// Core §2.2 lifecycle family, top tier: modes + cascade (§3.4/§3.7), Start/Stop
// mapped onto the §6.1 run command (§6 intro), the step chain (_M_SetStep/_M_Await,
// §6.5/§6.9(b)), the stall walk as a PENDING reason with instant rollup on an
// awaited module's Error (§6.9/§8.2), the §8.11.4 profiler wired in, and
// Starved/Blocked derived from the step's time class (§8.11.4(f)/§8.11.3).
// A Unit type overrides _M_Dispatch (its mode chain) + _M_Supports (+ §3.14 hooks).
FUNCTION_BLOCK ABSTRACT FB_UnitBase EXTENDS FB_CompositeModuleBase IMPLEMENTS I_Unit, I_SequenceHost
VAR_INPUT
    DecisionAnswer : INT;              // §6.11: chosen option index (0 = none yet)
    ReqControlOn   : BOOL;             // §9.8 HMI/data request; edge-consumed and access-gated
    ReqControlOff  : BOOL;
    HmiRequest     : ST_HmiRequest;     // §3.10/§14: arguments first, Sequence last
    {attribute 'OPC.UA.DA' := '0'}
    ControlDomain  : ST_ControlDomainStatus; // §9.8: optional shared cell/cage arrangement
END_VAR
VAR_OUTPUT
    Starved : BOOL;                    // §8.11.3 — derived from CurrentStep.TimeClass
    Blocked : BOOL;
    Domain  : ST_ControlDomainStatus;  // §9.8 read-only publication of the assigned domain
    ControlOnRequest  : BOOL;          // one-scan request to the owning domain coordinator
    ControlOffRequest : BOOL;
END_VAR
VAR_OUTPUT
    Profiler    : FB_CycleProfiler;    // §8.11.4 — HMI chart source
    CurrentStep : ST_StepRecord;       // §6.5 — feeds §6.9 walk AND the profiler
    // §3.13 sequence flow chart. Discovered from _M_SetStep, so a chain author
    // writes nothing; SequenceStepCount is the published length (§8.4 bounded).
    SequenceSteps : ARRAY[1..PL_Fraktal.MAX_SEQUENCE_STEPS] OF ST_SequenceStep;
    // §3.10.2 — the static half of each row: discovered once, never changes, so it
    // stays OFF the cyclic tree and is served through the config manifest under the
    // SAME browse paths as the live half (M_AppendConfig below).
    {attribute 'OPC.UA.DA' := '0'}
    SequenceStepDef : ARRAY[1..PL_Fraktal.MAX_SEQUENCE_STEPS] OF ST_SequenceStepDef;
    // §3.13 — which row each concurrent leg is running. Indexed by branch (0 = the
    // main line), so it is ~10 entries however long the chain is, and cheap enough
    // to stay in the cyclic read: the chart is right the moment its tab opens.
    ActiveSteps : ARRAY[0..PL_Fraktal.MAX_PARALLEL_BRANCHES] OF ST_SequenceCursor;
    // §6.9 — the errors and messages currently attached to rows. Sparse, so a small
    // table instead of 633 bytes reserved on every row for the usually-empty case.
    SequenceAnnotations : ARRAY[1..PL_Fraktal.MAX_SEQUENCE_ANNOTATIONS] OF ST_SequenceAnnotation;
    SequenceAnnotationCount : INT;
    SequenceStepCount : INT;
    CurrentStepElapsed : TIME;         // how long the active step has been running
    CurrentStepTimedOut : BOOL;        // active step outran its guard (§6.9 stall)

    Pending     : ST_Diagnostic;       // live stall reason (Low) — NOT a fault (§6.9)
    Decision    : ST_DecisionRequest;  // §6.11 active request ('' Prompt = none)
    {attribute 'OPC.UA.DA' := '0'}
    StallTime   : TIME := T#30S;       // guard when the step declares no ExpectedTime
    Model       : ST_ModelId;          // §3.1b active model identity (published for HMI/MES/trace)
    // §3.10.2 — static catalogs served via the QUERY_CONFIG manifest, not cyclically
    {attribute 'OPC.UA.DA' := '0'}
    AvailableModelCount : INT;         // §3.8 optional discoverable model/recipe catalog
    {attribute 'OPC.UA.DA' := '0'}
    AvailableModels : ARRAY[1..PL_Fraktal.MAX_RECIPES] OF ST_ModelId;
    Part        : ST_PartContext;      // §3.16.1 live part context (Present=FALSE, Uid='' = none)
    AlarmLog    : FB_AlarmLog;         // §8.3 — active list + closed ring + Blocking
    HostEvents  : FB_HostEventPublisher; // §11.6 fixed, bounded L3/MES projection
    Access      : FB_AccessManager;    // §7.7 — per-root session/policy (default: fully open)
    GoodCount   : UDINT;               // §8.11.2 — cycle verdict counters
    NokCount    : UDINT;
    ReworkCount : UDINT;
    NokReason   : E_Reason;            // §8.11.2 — last NOK's first-out attribution
    MachineState : E_MachineState;     // §8.11.3 — classified every scan (OEE/PackML/host)
    History     : ARRAY[1..PL_Fraktal.MAX_DIAG_RING] OF ST_Diagnostic;  // §6.9(a) ring (newest at HistoryHead)
    HistoryHead : INT;
    {attribute 'OPC.UA.DA' := '0'}
    ModePolicy  : ARRAY[0..PL_Fraktal.MODE_COUNT-1] OF ST_ModePolicy;    // §3.4.1 per-mode switch policy (station cfg; manifest-served)
    RunStyle    : E_RunStyle;          // §3.4.2 active run style (HMI-selectable; CONTINUOUS default)
    Oee         : ST_Oee;              // §8.5.1 accumulators + snapshot (published)
    // §8.5.2 - shifts, when a line is referenced (SetLine). 0 = no shift accounting.
    CurrentShift          : INT;
    ShiftStartedAt        : DT;
    ShiftHistory          : ARRAY[1..PL_Fraktal.MAX_SHIFT_HISTORY] OF ST_ShiftRecord; // newest first
    ShiftHistoryCount     : INT;
    ShiftHistoryTruncated : BOOL;
    OeeTrend    : ARRAY[1..PL_Fraktal.MAX_OEE_SAMPLES] OF ST_OeeSample; // §8.5.1 ring
    OeeTrendHead: INT;                 // newest sample index (0 = none yet)
    HmiResponse : ST_HmiResponse;
    ConfigRev   : UDINT;                // §3.10.2 manifest revision — HMI refetches on change
    // §3.8b — is this station's configuration actually SAFE? Transport
    // acknowledgement and Accepted mean a value is LIVE; this says whether it is
    // DURABLE, whether anything was lost at the last restart, and what the last
    // set operation did. Published cyclically because the answer changes without
    // anybody asking, and because it has to be visible BEFORE the restart that
    // would otherwise reveal it.
    ConfigPersist : ST_ConfigPersistStatus;
    // §3.8b — the store's set listing, refreshed on a LIST_CONFIG_SETS request.
    // Published, and read ON DEMAND: a client target-reads it when a set dialog
    // opens, never in its cyclic snapshot (§1.1 O4). It was marked DA := '0' until
    // 2026-09-27, which made the listing and the export lines unreachable over OPC
    // UA altogether - a client could request them and never read the answer.
    ConfigSets : ARRAY[1..PL_Fraktal.MAX_CONFIG_SETS] OF ST_ConfigSetInfo;
    ConfigSetCount : INT;
    // §3.8b — one line of a set's JSON document, served by EXPORT_CONFIG_SET.
    // Line 0 is the header and 1..RecordCount are the records, so a client pulls
    // a movable document a line at a time without a full buffer in the PLC —
    // the same paging discipline QUERY_CONFIG already uses.
    ConfigSetDocument : STRING(480);
    ConfigSetDocumentLine : INT;
    ConfigSetDocumentLines : INT;
    ModeActivePublished : E_Mode;       // properties are not OPC UA-visible
    RunningPublished : BOOL;
    StopPendingPublished : BOOL;
    SupportedModesPublished : ARRAY[0..PL_Fraktal.MODE_COUNT-1] OF BOOL;
    SupportedRunStylesPublished : ARRAY[0..2] OF BOOL;
    SystemHealth : ST_SystemHealthStatus; // §2.7/§8.12 live, trendable health
    SignalTower  : ST_SignalTowerOut;     // §8.13 single reusable mapping
END_VAR
VAR PERSISTENT
    // §3.8a station-config backing for the manifest-served ModePolicy output.
    // Version 0/unrecognized initializes safe defaults exactly once.
    _modePolicyVersion : UINT;
    _modePolicyStored : ARRAY[0..PL_Fraktal.MODE_COUNT-1] OF ST_ModePolicy;
END_VAR
VAR
    _fTrig    : R_TRIG;
    _mode     : E_Mode;
    _modeReq  : E_Mode;
    _modePend : BOOL;
    _modeExitFirst : BOOL;
    _stopReq  : BOOL;
    {attribute 'OPC.UA.DA' := '0'}
    _awaits   : I_Module;              // module the current step awaits (0 = none)
    _faultEvt : INT;                   // open ERROR event slot in AlarmLog (0 = none)
    _tStall   : TON;
    _seqIndex : INT;                   // row recorded LAST, i.e. the step action running now
    _stepSinceMs : DWORD;              // monotonic start of the main-line step
    // §6.12 — per-row clock and liveness. With a parallel step several rows are
    // active at once, so one cursor is no longer enough to say what is running or
    // for how long. Bounded exactly like the row table itself (§1.1 O10).
    // Per-LEG, not per row: a leg has one active step, so the per-scan sweep is ~10
    // iterations instead of up to MAX_SEQUENCE_STEPS.
    _branchSinceMs : ARRAY[0..PL_Fraktal.MAX_PARALLEL_BRANCHES] OF DWORD;
    _branchTouched : ARRAY[0..PL_Fraktal.MAX_PARALLEL_BRANCHES] OF BOOL;
    _tDecision: TON;                   // §6.11 monotonic active-decision timeout
    _decisionConflictLogged : BOOL;    // one audit record per conflicting request
    _decisionResolutionLogged : BOOL;  // operator/timeout resolution logged once
    _stepReq  : BOOL;                  // §3.4.2 pending single-step request (edge-consumed)
    _holdRun  : BOOL;                  // §3.4.2 HOLD_TO_RUN input held (NON-SAFETY, §9)
    _stepArm  : R_TRIG;
    _errClr   : R_TRIG;                // §6.9 the ERROR state ended
    _oeeLast  : TIME;                  // §8.5.1 last accumulation stamp
    _oeeSampMs: UDINT;                 // ms since last trend sample
    // §8.5.2 shift accounting
    {attribute 'OPC.UA.DA' := '0'}
    _pLine : POINTER TO FB_LineData;
    // §3.8a - model data: the provider and key of this root's own recipe record,
    // and the buffer a model-scoped request loads another model's record into.
    {attribute 'OPC.UA.DA' := '0'}
    _modelProvider : I_RecipeProvider;
    _modelKey : STRING(80);
    _viewModelCode : STRING(64);
    {attribute 'OPC.UA.DA' := '0'}
    _modelBuf : ARRAY[1..PL_Fraktal.MAX_MODEL_DATA_BYTES] OF BYTE;
    _lineHost : BOOL;                  // §3.8e this root ticks the line it references
    _lineRevSeen : UDINT;              // §3.8e line revision last reflected in ConfigRev
    _shiftInit : BOOL;
    _shiftSync : BOOL;
    _shiftManualReset : BOOL;
    _hmiLastSequence : UDINT;
    {attribute 'OPC.UA.DA' := '0'}
    _configPager : FB_ConfigPager;     // §3.10.2 QUERY_CONFIG window writer
    // §3.8b — the parameter-set store. Absent (the shipped default for a Unit
    // nobody wired one into) means save/load/list are simply not offered, which
    // is published as StorePresent = FALSE rather than failing at the first
    // request an operator makes.
    {attribute 'OPC.UA.DA' := '0'}
    _configStore : I_ConfigStore;
    // §3.8b durability. _persistWriter is the shipped LOCAL_RETAIN default and
    // is used unless a deployment injects something else, so a conforming
    // station persists its parametrization with no file system, no network and
    // no configuration — and with no line of project code either (§1.1 O1).
    {attribute 'OPC.UA.DA' := '0'}
    _persistWriter : FB_PersistentDataWriter;
    {attribute 'OPC.UA.DA' := '0'}
    _persistence : I_ConfigPersistence;
    _persistSinceMs : DWORD;           // monotonic ms the current window started at
    _persistEvt : INT;                 // open PersistFailed event slot (0 = none)
    _restoreEvt : INT;                 // open restore-loss event slot (0 = none)
    {attribute 'OPC.UA.DA' := '0'}
    _setJson : FB_ConfigSetJson;       // §3.8b text projection (export/import)
    _importOpen : BOOL;                // an IMPORT_CONFIG_SET save is in progress
    // §3.8b - a set line arriving in pieces (IMPORT_CONFIG_SET, IntValue = 1).
    // A request carries 255 characters and a line may hold 480, so the HMI
    // splits it; the pieces are joined here, and nowhere else.
    {attribute 'OPC.UA.DA' := '0'}
    _importPart : STRING(480);
    // §7.6.1a hold-to-run. The request is LATCHED and re-asserted every scan,
    // because a mailbox delivers one request per sequence and the axis expects
    // to be asked every scan it should keep moving. The latch is what makes
    // that work over a transport; the deadline is what keeps it safe, since a
    // client that stops refreshing - closed, crashed, unplugged - lets the hold
    // expire instead of leaving the machine moving.
    _heldPath  : STRING(255);
    _heldValue : DINT;
    _heldActive : BOOL;
    _heldSinceMs : DWORD;
    // §3.13 - the flow chart changed and the manifest revision owes it a bump.
    // Held until the growth settles, so one burst of row discovery costs one
    // refetch instead of one per row (PL_Fraktal.CHART_REV_SETTLE_MS).
    _chartDirty : BOOL;
    _chartTouchedMs : DWORD;
    {attribute 'OPC.UA.DA' := '0'}
    _carrier  : I_PartCarrier;         // §3.16.2 injected part carrier (0 = traceability off)
    {attribute 'OPC.UA.DA' := '0'}
    _healthPublisher : FB_SystemHealthPublisher;
    {attribute 'OPC.UA.DA' := '0'}
    _healthInput : ST_SystemHealthInput;
    {attribute 'OPC.UA.DA' := '0'}
    _healthParCfg : ST_SystemHealthParCfg;
    _healthConfigured : BOOL;
    {attribute 'OPC.UA.DA' := '0'}
    _towerMapper : FB_SignalTower;
    {attribute 'OPC.UA.DA' := '0'}
    _towerParCfg : ST_SignalTowerParCfg;
    _lampTestRequest : BOOL;
    {attribute 'OPC.UA.DA' := '0'}
    _sequences : ARRAY[1..PL_Fraktal.MAX_SEQUENCES] OF I_Sequence;
    _sequenceCount : INT;
    // §7.5 commissioning/engineering gate register, injected by the composition
    // root. Absent (the shipped default) = a production image: no gate is
    // annunciated and ForceChannel refuses every request (fail closed).
    {attribute 'OPC.UA.DA' := '0'}
    _engineering : REFERENCE TO FB_EngineeringMode;
    // §7.5.2 open standing event per registered gate (0 = none open yet)
    _engineeringEvt : ARRAY[1..PL_Fraktal.MAX_ENGINEERING_GATES] OF INT;
END_VAR
VAR CONSTANT
    // §3.8b — layout version of the retained ModePolicy image. Bump it when a
    // member is added to ST_ModePolicy or the array is resized; the retained
    // image is then rejected and annunciated instead of read by field position.
    MODE_POLICY_SCHEMA : UINT := 1;
    // §3.8b — schema version stamped into every set this root produces, so a set
    // document that outlives the build that wrote it can be recognized rather
    // than guessed at (§13).
    CONFIG_SET_SCHEMA : UINT := 1;
END_VAR

Cyclic();

// Core §7.8 helper — append one non-interlock reason (bounds-checked).
METHOD PROTECTED _M_AddReason
VAR_IN_OUT
    Report : ST_ReleaseReport;
END_VAR
VAR_INPUT
    Text : STRING(255);
    Reason : E_Reason;
    Kind : E_ReleaseKind;
END_VAR
IF Report.Count >= PL_Fraktal.MAX_RELEASE_REASONS THEN
    RETURN;
END_IF
Report.Count := Report.Count + 1;
Report.Reasons[Report.Count].Description := Text;
Report.Reasons[Report.Count].ReasonCode  := Reason;
Report.Reasons[Report.Count].SourcePath  := _name;
Report.Reasons[Report.Count].Kind        := Kind;
Report.Reasons[Report.Count].Bypassable  := FALSE;
END_METHOD

// Core §7.8 — concrete Units override to append the active mode's immediate
// entry/frontier records via PermIntlk.AppendFailed(SourcePath, Report). Future step waits
// stay in CurrentStep/Pending and are not blanket Start conditions. Base: nothing.
METHOD PROTECTED _M_AppendInterlocks
VAR_IN_OUT
    Report : ST_ReleaseReport;
END_VAR
;
END_METHOD

// Core §7.8 — target-aware hook for the MANUAL release rollup: a concrete Unit
// overrides to append the §7.6 Release<Function> conditions of the SPECIFIC target
// module. Base delegates to the Unit-level hook (non-breaking default).
METHOD PROTECTED _M_AppendManualInterlocks
VAR_INPUT
    TargetPath : STRING(255);
    Value : DINT;
END_VAR
VAR_IN_OUT
    Report : ST_ReleaseReport;
END_VAR
_M_AppendInterlocks(Report := Report);
END_METHOD

// §6.11 option-aware release seam. The base validates session, active prompt and
// option identity; a concrete Unit appends the ordinary process conditions that a
// "continue"-style option must satisfy. Safety and child interlocks still remain
// authoritative at their owning modules.
METHOD PROTECTED _M_AppendDecisionInterlocks
VAR_INPUT
    Option : INT;
END_VAR
VAR_IN_OUT
    Report : ST_ReleaseReport;
END_VAR
;
END_METHOD

// §6.11 — publish a typed decision request (single active slot)
METHOD PROTECTED _M_AskDecision
VAR_INPUT
    Req : ST_DecisionRequest;
END_VAR
VAR
    candidate : ST_DecisionRequest;
END_VAR
candidate := Req;
IF candidate.SourcePath = '' THEN
    candidate.SourcePath := _name;
END_IF
// A sequence presents the same request every scan while its step waits. That is
// idempotent. A different producer never overwrites the visible active request.
IF Decision.Prompt <> '' THEN
    IF _M_DecisionMatches(Req := candidate) THEN
        RETURN;
    END_IF
    IF NOT _decisionConflictLogged THEN
        _M_LogDecision(EventKey := 'std.audit.decisionOverlapRejected',
            SourcePath := candidate.SourcePath, Option := 0);
        _decisionConflictLogged := TRUE;
    END_IF
    RETURN;
END_IF
IF NOT _M_ValidateDecision(Req := candidate) THEN
    _M_LogDecision(EventKey := 'std.audit.decisionInvalidRejected',
        SourcePath := candidate.SourcePath, Option := candidate.Default);
    _M_Fault(E_Reason.UNSUPPORTED_COMMAND, 'std.error.invalidDecisionRequest');
    RETURN;
END_IF
Decision := candidate;
DecisionAnswer := 0;
_decisionConflictLogged := FALSE;
_decisionResolutionLogged := FALSE;
_tDecision(IN := FALSE);
_M_LogDecision(EventKey := 'std.audit.decisionRequested',
    SourcePath := Decision.SourcePath, Option := 0);
END_METHOD

// Clear the complete public slot and all private latches atomically.
METHOD PRIVATE _M_ClearDecisionState
VAR
    i : INT;
END_VAR
_tDecision(IN := FALSE);
DecisionAnswer := 0;
Decision.Prompt := '';
Decision.Default := 0;
Decision.Timeout := T#0S;
Decision.SourcePath := '';
FOR i := 1 TO PL_Fraktal.MAX_OPTIONS DO
    Decision.Options[i] := '';
END_FOR
_decisionConflictLogged := FALSE;
_decisionResolutionLogged := FALSE;
END_METHOD

// §6.11 one-slot resolver. Operator input wins if it is accepted in the same scan
// the timeout expires; _M_HandleHmiRequest runs immediately before this method.
METHOD PRIVATE _M_DecisionCyclic
IF _exec <> E_ExecState.BUSY THEN
    IF Decision.Prompt <> '' THEN
        _M_LogDecision(EventKey := 'std.audit.decisionWithdrawn',
            SourcePath := Decision.SourcePath, Option := 0);
        _M_ClearDecisionState();
    ELSE
        _tDecision(IN := FALSE);
    END_IF
    RETURN;
END_IF
IF Decision.Prompt = '' THEN
    _tDecision(IN := FALSE);
    RETURN;
END_IF
IF DecisionAnswer <> 0 THEN
    _tDecision(IN := FALSE);
    IF (DecisionAnswer < 1) OR (DecisionAnswer > PL_Fraktal.MAX_OPTIONS) THEN
        _M_LogDecision(EventKey := 'std.audit.decisionAnswerRejected',
            SourcePath := Decision.SourcePath, Option := DecisionAnswer);
        DecisionAnswer := 0;
        RETURN;
    END_IF
    IF Decision.Options[DecisionAnswer] = '' THEN
        _M_LogDecision(EventKey := 'std.audit.decisionAnswerRejected',
            SourcePath := Decision.SourcePath, Option := DecisionAnswer);
        DecisionAnswer := 0;
        RETURN;
    END_IF
    IF NOT _decisionResolutionLogged THEN
        _M_LogDecision(EventKey := 'std.audit.decisionOperatorResolved',
            SourcePath := Decision.SourcePath, Option := DecisionAnswer);
        _decisionResolutionLogged := TRUE;
    END_IF
    RETURN;
END_IF
IF Decision.Timeout <= T#0S THEN
    _tDecision(IN := FALSE);
    RETURN;
END_IF
_tDecision(IN := TRUE, PT := Decision.Timeout);
IF _tDecision.Q THEN
    DecisionAnswer := Decision.Default;             // validated when accepted
    _tDecision(IN := FALSE);
    _M_LogDecision(EventKey := 'std.audit.decisionTimeoutResolved',
        SourcePath := Decision.SourcePath, Option := DecisionAnswer);
    _decisionResolutionLogged := TRUE;
END_IF
END_METHOD

// Full value comparison makes repeated presentation idempotent while treating a
// changed option/default/timeout as a different request that must not overwrite.
METHOD PRIVATE _M_DecisionMatches : BOOL
VAR_INPUT
    Req : ST_DecisionRequest;
END_VAR
VAR
    i : INT;
END_VAR
_M_DecisionMatches := FALSE;
IF (Decision.Prompt <> Req.Prompt)
OR (Decision.Default <> Req.Default)
OR (Decision.Timeout <> Req.Timeout)
OR (Decision.SourcePath <> Req.SourcePath) THEN
    RETURN;
END_IF
FOR i := 1 TO PL_Fraktal.MAX_OPTIONS DO
    IF Decision.Options[i] <> Req.Options[i] THEN
        RETURN;
    END_IF
END_FOR
_M_DecisionMatches := TRUE;
END_METHOD

// Domain audit: request, rejection and resolution are closed MESSAGE events.
METHOD PRIVATE _M_LogDecision
VAR_INPUT
    EventKey : STRING(160);
    SourcePath : STRING(255);
    Option : INT;
END_VAR
VAR
    slot : INT;
    textValue : STRING(255);
    sourceValue : STRING(255);
END_VAR
textValue := EventKey;
IF Option <> 0 THEN
    textValue := CONCAT(textValue, ' option=');
    textValue := CONCAT(textValue, TO_STRING(Option));
END_IF
sourceValue := SourcePath;
IF sourceValue = '' THEN
    sourceValue := _name;
END_IF
slot := AlarmLog.Raise(Reason := E_Reason.NONE, Text := textValue,
    Source := sourceValue, Severity := E_Severity.LOW,
    Category := E_Category.PROCESS, ResetClass := E_ResetClass.AUTO_RESET);
IF slot > 0 THEN
    AlarmLog.Gone(Slot := slot);
END_IF
END_METHOD

// A finite timeout requires a real safe default. An indefinite request may omit
// Default, but every published request still needs at least one selectable option.
METHOD PRIVATE _M_ValidateDecision : BOOL
VAR_INPUT
    Req : ST_DecisionRequest;
END_VAR
VAR
    i : INT;
    hasOption : BOOL;
END_VAR
_M_ValidateDecision := FALSE;
IF (Req.Prompt = '') OR (Req.Timeout < T#0S) THEN
    RETURN;
END_IF
hasOption := FALSE;
FOR i := 1 TO PL_Fraktal.MAX_OPTIONS DO
    IF Req.Options[i] <> '' THEN
        hasOption := TRUE;
    END_IF
END_FOR
IF NOT hasOption THEN
    RETURN;
END_IF
IF (Req.Timeout > T#0S) OR (Req.Default <> 0) THEN
    IF (Req.Default < 1) OR (Req.Default > PL_Fraktal.MAX_OPTIONS) THEN
        RETURN;
    END_IF
    IF Req.Options[Req.Default] = '' THEN
        RETURN;
    END_IF
END_IF
_M_ValidateDecision := TRUE;
END_METHOD

// §6.9(b) — named plain-condition wait; returns the condition so steps read naturally
METHOD PROTECTED _M_Await : BOOL
VAR_INPUT
    Idx   : INT;
    Label : STRING(120);
    Ok    : BOOL;
END_VAR
IF (Idx >= 1) AND (Idx <= PL_Fraktal.MAX_STEP_CONDS) THEN
    CurrentStep.Conds[Idx].Label := Label;
    CurrentStep.Conds[Idx].Ok    := Ok;
END_IF
_M_Await := Ok;
END_METHOD

// §3.7 — offer the mode to child Units; a child may reject (graceful)
METHOD PROTECTED _M_CascadeMode
VAR_INPUT
    Mode : E_Mode;
END_VAR
VAR
    i  : INT;
    iu : I_Unit;
END_VAR
FOR i := 1 TO _nChild DO
    IF _children[i] <> 0 THEN
        IF __QUERYINTERFACE(_children[i], iu) THEN   // [TC3] capability query — TC3 §3.2
            iu.SetMode(Mode);
        END_IF
    END_IF
END_FOR
END_METHOD

METHOD PROTECTED _M_ClearPending
Pending.ReasonCode  := E_Reason.NONE;
Pending.Description := '';
Pending.TimeSynchronized := FALSE;
END_METHOD

// §14.3 security audit for accepted remote mutations. Operational methods may
// additionally emit their domain event (manual action, OEE reset, shelving); this
// record supplies the remote request kind and authenticated user without secrets.
METHOD PROTECTED _M_AuditHmiAccepted
VAR_INPUT
    Kind : E_HmiRequestKind;
    TargetPath : STRING(255);
    Accepted : BOOL;
END_VAR
VAR
    auditable : BOOL;
    auditSlot : INT;
    textValue : STRING(255);
    sourcePath : STRING(255);
END_VAR
IF NOT Accepted THEN
    RETURN;
END_IF
CASE Kind OF
    E_HmiRequestKind.SET_MODE, E_HmiRequestKind.SET_MODEL,
    E_HmiRequestKind.START, E_HmiRequestKind.STOP,
    E_HmiRequestKind.CONTROL_ON, E_HmiRequestKind.CONTROL_OFF,
    E_HmiRequestKind.OPERATOR_RESET, E_HmiRequestKind.DECISION_ANSWER,
    E_HmiRequestKind.MANUAL_COMMAND, E_HmiRequestKind.SET_RUN_STYLE,
    E_HmiRequestKind.STEP_REQUEST, E_HmiRequestKind.SET_HOLD_RUN,
    E_HmiRequestKind.RESET_OEE, E_HmiRequestKind.WRITE_CONFIG,
    E_HmiRequestKind.SHELVE_ALARM, E_HmiRequestKind.UNSHELVE_ALARM,
    E_HmiRequestKind.FORCE_CHANNEL, E_HmiRequestKind.SET_ACCESS_LEVEL,
    E_HmiRequestKind.SET_SESSION_TIMEOUT, E_HmiRequestKind.LAMP_TEST,
    E_HmiRequestKind.CAPTURE_CONFIG, E_HmiRequestKind.SAVE_CONFIG_SET,
    E_HmiRequestKind.LOAD_CONFIG_SET, E_HmiRequestKind.ACK_CONFIG_RESTORE,
    E_HmiRequestKind.IMPORT_CONFIG_SET, E_HmiRequestKind.DELETE_CONFIG_SET,
    E_HmiRequestKind.SET_CLASS_LEVEL:
        auditable := TRUE;
ELSE
    auditable := FALSE;
END_CASE
IF NOT auditable THEN
    RETURN;
END_IF
Access.RecordActivity();
textValue := CONCAT('std.audit.hmiAccepted kind=', TO_STRING(TO_DINT(Kind)));
textValue := CONCAT(textValue, ' user=');
textValue := CONCAT(textValue, Access.CurrentUser);
// §3.8b — a set operation is audited WITH the set name and record count: "the
// operator loaded a set" is not an audit record anyone can act on later.
IF (Kind = E_HmiRequestKind.SAVE_CONFIG_SET)
OR (Kind = E_HmiRequestKind.LOAD_CONFIG_SET)
OR (Kind = E_HmiRequestKind.DELETE_CONFIG_SET) THEN
    textValue := CONCAT(textValue, ' set=');
    textValue := CONCAT(textValue, ConfigPersist.LastSetName);
    textValue := CONCAT(textValue, ' records=');
    textValue := CONCAT(textValue, INT_TO_STRING(ConfigPersist.LastSetRecords));
END_IF
sourcePath := TargetPath;
IF sourcePath = '' THEN
    sourcePath := _name;
END_IF
auditSlot := AlarmLog.Raise(Reason := E_Reason.NONE, Text := textValue,
    Source := sourcePath, Severity := E_Severity.LOW, Category := E_Category.SYSTEM,
    ResetClass := E_ResetClass.AUTO_RESET);
IF auditSlot > 0 THEN AlarmLog.Gone(Slot := auditSlot); END_IF
END_METHOD

// Module paths are qualified dotted Fraktal identities (§4.8). A request routed
// through this root may target the root itself or one descendant, never a peer.
METHOD PRIVATE _M_OwnsModulePath : BOOL
VAR_INPUT
    Path : STRING(255);
END_VAR
VAR
    prefix : STRING(255);
END_VAR
prefix := CONCAT(_name, '.');
_M_OwnsModulePath := (Path = _name) OR (FIND(Path, prefix) = 1);
END_METHOD

// call at the finish step (§8.11.1): publishes the profile; FALSE = stop granted
METHOD PROTECTED _M_EndOfCycle : BOOL
Profiler.CycleComplete();
IF _stopReq THEN
    _stopReq := FALSE;
    Execute := FALSE;
    _M_Complete();
    _M_EndOfCycle := FALSE;
ELSE
    _M_EndOfCycle := TRUE;
END_IF
END_METHOD

// §3.10/§14 — consume one committed OPC UA request exactly once.
METHOD PROTECTED _M_HandleHmiRequest
VAR
    modelId  : ST_ModelId;
    modeReq  : E_Mode;
    styleReq : E_RunStyle;
    gateReq  : E_GatedAction;
    levelReq : E_AccessLevel;
    alarmSlot : INT;
    policyValueValid : BOOL;
    configKindReq : E_ConfigKind;
END_VAR
IF HmiRequest.Sequence = _hmiLastSequence THEN
    RETURN;
ELSE
    _hmiLastSequence := HmiRequest.Sequence;
END_IF

HmiResponse.Accepted := FALSE;
HmiResponse.Diagnostic := '';
HmiResponse.Report.Count := 0;
HmiResponse.Report.Released := FALSE;
// A held line piece belongs to the very next import request. Anything else in
// between means the line was abandoned, so it is dropped rather than glued to
// whatever arrives later.
IF HmiRequest.Kind <> E_HmiRequestKind.IMPORT_CONFIG_SET THEN
    _importPart := '';
END_IF

CASE HmiRequest.Kind OF
    E_HmiRequestKind.LOGIN:
        HmiResponse.Accepted := Access.RequestLogin(User := HmiRequest.User, Secret := HmiRequest.Secret);
    E_HmiRequestKind.LOGOUT:
        HmiResponse.Accepted := Access.RequestLogout();
    E_HmiRequestKind.SET_MODE:
        IF (HmiRequest.IntValue >= 0) AND (HmiRequest.IntValue < PL_Fraktal.MODE_COUNT) THEN
            modeReq := HmiRequest.IntValue;
            HmiResponse.Accepted := SetMode(Mode := modeReq);
        ELSE
            HmiResponse.Diagnostic := 'std.error.unsupportedModeRequest';
        END_IF
    E_HmiRequestKind.SET_MODEL:
        modelId.ModelCode := HmiRequest.TextValue;
        HmiResponse.Accepted := SetModel(Id := modelId);
    E_HmiRequestKind.START:
        HmiResponse.Accepted := Start();
    E_HmiRequestKind.STOP:
        HmiResponse.Accepted := Stop();
    E_HmiRequestKind.CONTROL_ON:
        HmiResponse.Accepted := RequestControlPower(ControlOn := TRUE);
    E_HmiRequestKind.CONTROL_OFF:
        HmiResponse.Accepted := RequestControlPower(ControlOn := FALSE);
    E_HmiRequestKind.OPERATOR_RESET:
        HmiResponse.Accepted := OperatorReset();
    E_HmiRequestKind.DECISION_ANSWER:
        HmiResponse.Accepted := SubmitDecision(Option := TO_INT(HmiRequest.IntValue),
            Report := HmiResponse.Report);
    E_HmiRequestKind.MANUAL_COMMAND:
        HmiResponse.Accepted := ManualCommandTo(TargetPath := HmiRequest.TargetPath, Value := HmiRequest.IntValue);
    E_HmiRequestKind.MANUAL_HELD:
        HmiResponse.Accepted := ManualHeldTo(TargetPath := HmiRequest.TargetPath,
            Value := HmiRequest.IntValue, Held := HmiRequest.BoolValue);
    E_HmiRequestKind.SET_RUN_STYLE:
        IF (HmiRequest.IntValue >= 0) AND (HmiRequest.IntValue <= 2) THEN
            styleReq := HmiRequest.IntValue;
            HmiResponse.Accepted := SetRunStyle(Style := styleReq);
        ELSE
            HmiResponse.Diagnostic := 'std.error.unsupportedRunStyleRequest';
        END_IF
    E_HmiRequestKind.STEP_REQUEST:
        HmiResponse.Accepted := StepRequest();
    E_HmiRequestKind.SET_HOLD_RUN:
        HmiResponse.Accepted := SetHoldRun(Held := HmiRequest.BoolValue);
    E_HmiRequestKind.RELEASE_START:
        ReleaseReportStart(Report := HmiResponse.Report);
        HmiResponse.Accepted := TRUE;
    E_HmiRequestKind.RELEASE_MANUAL:
        ReleaseReportManual(TargetPath := HmiRequest.TargetPath, Value := HmiRequest.IntValue,
            Report := HmiResponse.Report);
        HmiResponse.Accepted := TRUE;
    E_HmiRequestKind.RELEASE_ACTION:
        IF (HmiRequest.IntValue >= 0)
        AND (HmiRequest.IntValue <= TO_DINT(E_GatedAction.CONFIG_SET)) THEN
            gateReq := HmiRequest.IntValue;
            ReleaseReportAction(Gate := gateReq, Report := HmiResponse.Report);
            HmiResponse.Accepted := TRUE;
        ELSE
            HmiResponse.Diagnostic := 'std.error.unsupportedGatedActionRequest';
        END_IF
    E_HmiRequestKind.RESET_OEE:
        HmiResponse.Accepted := ResetOee();
    E_HmiRequestKind.WRITE_CONFIG:
        // §3.8a - DurationMs names the model a model-data write is for
        // (0 = the active model, n = AvailableModels[n]); other values ignore it.
        HmiResponse.Accepted := WriteModelConfig(ModelIndex := HmiRequest.DurationMs,
            TargetPath := HmiRequest.TargetPath, WriteKey := HmiRequest.NameValue,
            Revision := HmiRequest.IntValue, TextValue := HmiRequest.TextValue);
    E_HmiRequestKind.SHELVE_ALARM:
        alarmSlot := AlarmLog.FindActiveSlot(SourcePath := HmiRequest.TargetPath,
            Description := HmiRequest.TextValue);
        IF alarmSlot > 0 THEN
            HmiResponse.Accepted := ShelveAlarm(Slot := alarmSlot,
                DurationS := HmiRequest.DurationMs / 1000);
        ELSE
            HmiResponse.Diagnostic := 'std.error.alarmIdentityNotUnique';
        END_IF
    E_HmiRequestKind.UNSHELVE_ALARM:
        alarmSlot := AlarmLog.FindActiveSlot(SourcePath := HmiRequest.TargetPath,
            Description := HmiRequest.TextValue);
        IF alarmSlot > 0 THEN
            HmiResponse.Accepted := UnshelveAlarm(Slot := alarmSlot);
        ELSE
            HmiResponse.Diagnostic := 'std.error.alarmIdentityNotUnique';
        END_IF
    E_HmiRequestKind.FORCE_CHANNEL:
        HmiResponse.Accepted := ForceChannel(ChannelPath := HmiRequest.TargetPath,
            Force := HmiRequest.BoolValue, BoolText := HmiRequest.TextValue,
            AnalogText := HmiRequest.NameValue);
    E_HmiRequestKind.QUERY_CONFIG:
        // §3.10.2 — serve one manifest page: re-walk the deterministic export
        // enumeration, storing only the requested window (no full buffer).
        // §3.8d: no blanket DATA_READ refusal any more - a class may be readable
        // below it. Each entry is served with or without its value by its level.
        _configPager.M_SetAccess(pAccess := ADR(Access));
        // §3.8a - DurationMs names the model whose model-data values to serve.
        IF NOT _configPager.M_Setup(Target := ADR(HmiResponse.ConfigPage),
            PageIndex := TO_INT(HmiRequest.IntValue), Revision := ConfigRev) THEN
            HmiResponse.Diagnostic := 'std.error.hmiRequestRejected';
        ELSIF M_AppendModelConfig(Pager := _configPager,
                ModelIndex := HmiRequest.DurationMs) THEN
            _configPager.M_Finish();
            HmiResponse.Accepted := TRUE;
        ELSE
            HmiResponse.Diagnostic := 'std.error.modelNotAvailable';
        END_IF
    E_HmiRequestKind.SET_ACCESS_LEVEL:
        policyValueValid := TRUE;
        IF HmiRequest.TextValue = '0' THEN
            levelReq := E_AccessLevel.NONE;
        ELSIF HmiRequest.TextValue = '1' THEN
            levelReq := E_AccessLevel.OPERATOR;
        ELSIF HmiRequest.TextValue = '2' THEN
            levelReq := E_AccessLevel.TECHNICIAN;
        ELSIF HmiRequest.TextValue = '3' THEN
            levelReq := E_AccessLevel.ENGINEER;
        ELSIF HmiRequest.TextValue = '4' THEN
            levelReq := E_AccessLevel.ADMIN;
        ELSE
            policyValueValid := FALSE;
        END_IF
        IF policyValueValid
        AND (HmiRequest.IntValue >= 0)
        AND (HmiRequest.IntValue <= TO_DINT(E_GatedAction.CONFIG_SET)) THEN
            gateReq := HmiRequest.IntValue;
            HmiResponse.Accepted := SetAccessLevel(Gate := gateReq, Level := levelReq);
        ELSE
            HmiResponse.Diagnostic := 'std.error.accessPolicyValueInvalid';
        END_IF
    E_HmiRequestKind.SET_SESSION_TIMEOUT:
        HmiResponse.Accepted := SetSessionTimeout(TimeoutMs := HmiRequest.DurationMs);
    E_HmiRequestKind.LAMP_TEST:
        HmiResponse.Accepted := RequestLampTest();
    E_HmiRequestKind.CAPTURE_CONFIG:
        // §3.8c(a) — a capture is routed through the SAME acknowledged mailbox as
        // the typed write it replaces, with the same arguments minus the value:
        // the number comes from the machine, not from the client.
        HmiResponse.Accepted := CaptureConfig(TargetPath := HmiRequest.TargetPath,
            WriteKey := HmiRequest.NameValue, Revision := HmiRequest.IntValue);
    E_HmiRequestKind.SAVE_CONFIG_SET:
        IF (HmiRequest.IntValue >= 0)
        AND (HmiRequest.IntValue <= TO_DINT(E_ConfigKind.LINE_CFG)) THEN
            configKindReq := HmiRequest.IntValue;
            HmiResponse.Accepted := SaveConfigSet(SetName := HmiRequest.TextValue,
                Kind := configKindReq);
        ELSE
            HmiResponse.Diagnostic := 'std.error.configSetKindInvalid';
        END_IF
    E_HmiRequestKind.LOAD_CONFIG_SET:
        HmiResponse.Accepted := LoadConfigSet(SetName := HmiRequest.TextValue);
        IF NOT HmiResponse.Accepted THEN
            HmiResponse.Diagnostic := 'std.error.configSetRejected';
        END_IF
    E_HmiRequestKind.LIST_CONFIG_SETS:
        HmiResponse.Accepted := ListConfigSets();
    E_HmiRequestKind.ACK_CONFIG_RESTORE:
        HmiResponse.Accepted := AcknowledgeConfigRestore();
        IF NOT HmiResponse.Accepted THEN
            HmiResponse.Diagnostic := 'std.error.configRestoreAckRefused';
        END_IF
    E_HmiRequestKind.EXPORT_CONFIG_SET:
        HmiResponse.Accepted := ExportConfigSetLine(SetName := HmiRequest.TextValue,
            Line := TO_INT(HmiRequest.IntValue));
    E_HmiRequestKind.IMPORT_CONFIG_SET:
        HmiResponse.Accepted := ImportConfigSetPiece(Piece := HmiRequest.TextValue,
            More := HmiRequest.IntValue = 1, Commit := HmiRequest.BoolValue);
        IF NOT HmiResponse.Accepted THEN
            HmiResponse.Diagnostic := 'std.error.configSetLineRejected';
        END_IF
    E_HmiRequestKind.SET_CLASS_LEVEL:
        HmiResponse.Accepted := SetDataClassLevel(ClassId := HmiRequest.NameValue,
            Level := HmiRequest.IntValue, ForWrite := HmiRequest.BoolValue);
        IF NOT HmiResponse.Accepted THEN
            HmiResponse.Diagnostic := 'std.error.accessPolicyValueInvalid';
        END_IF
    E_HmiRequestKind.DELETE_CONFIG_SET:
        HmiResponse.Accepted := DeleteConfigSet(SetName := HmiRequest.TextValue);
        IF NOT HmiResponse.Accepted THEN
            HmiResponse.Diagnostic := 'std.error.configSetDeleteRefused';
        END_IF
    E_HmiRequestKind.NONE:
        HmiResponse.Diagnostic := 'std.error.emptyHmiRequest';
ELSE
    HmiResponse.Diagnostic := 'std.error.unsupportedHmiRequest';
END_CASE

IF NOT HmiResponse.Accepted AND (HmiResponse.Diagnostic = '') THEN
    HmiResponse.Diagnostic := 'std.error.hmiRequestRejected';
ELSE
    HmiResponse.Diagnostic := HmiResponse.Diagnostic;
END_IF
_M_AuditHmiAccepted(Kind := HmiRequest.Kind, TargetPath := HmiRequest.TargetPath,
    Accepted := HmiResponse.Accepted);
HmiRequest.Secret := '';
HmiResponse.AckSequence := _hmiLastSequence;
END_METHOD

// §11.6 one owning projection helper; callers supply only event-specific fields.
METHOD PRIVATE _M_HostEvent : BOOL
VAR_INPUT
    Kind          : E_HostEventKind;
    PartUid       : STRING(64);
    Subject       : STRING(80);
    Value         : STRING(80);
    Verdict       : E_Verdict;
    ReasonCode    : E_Reason;
END_VAR
_M_HostEvent := HostEvents.Emit(Kind := Kind,
    StationPath := _name, PartUid := PartUid, Subject := Subject,
    Value := Value, Verdict := Verdict, ReasonCode := ReasonCode);
END_METHOD

// §3.4.1/§3.14.4 — default per-mode switch policy. Station config (§3.8a) may
// overwrite ModePolicy[] after this. By FRAMEWORK DEFAULT a mode change while a
// sequence runs performs an IMMEDIATE software abort (E-stop-like, not a safety
// function, §3.14.4) — so Style defaults to IMMEDIATE. GRACEFUL completion is an
// opt-in: a Unit overrides OnModeExit to stop-after-cycle, or station config sets
// Style := GRACEFUL for a mode. Shield only governs acceptance while running.
METHOD PROTECTED _M_InitModePolicy
VAR
    i : INT;
END_VAR
FOR i := 0 TO PL_Fraktal.MODE_COUNT-1 DO
    ModePolicy[i].Shield := E_ModeSwitchShield.CONFIRM;
    ModePolicy[i].Style  := E_ModeSwitchStyle.IMMEDIATE;
END_FOR
// Setup modes a running machine may not leave without an explicit Stop first.
ModePolicy[TO_INT(E_Mode.CHANGEOVER)].Shield := E_ModeSwitchShield.BLOCKED_WHILE_RUNNING;
ModePolicy[TO_INT(E_Mode.CALIBRATION)].Shield:= E_ModeSwitchShield.BLOCKED_WHILE_RUNNING;
// HOME and MANUAL are freely interruptible; both inherit the IMMEDIATE default.
ModePolicy[TO_INT(E_Mode.HOME)].Shield       := E_ModeSwitchShield.INTERRUPTIBLE;
ModePolicy[TO_INT(E_Mode.MANUAL)].Shield     := E_ModeSwitchShield.INTERRUPTIBLE;
END_METHOD

// §8.5.1 — pure recompute of A/P/Q/OEE from the accumulators (testable in isolation).
// Invalid factors are OMITTED from the product, never assumed 100% (O7).
METHOD PROTECTED _M_OeeCompute
VAR
    total : UDINT;
    denomA: UDINT;
END_VAR
denomA := Oee.RunMs + Oee.DownMs;
Oee.AvailValid := denomA > 0;
IF Oee.AvailValid THEN
    Oee.Availability := UDINT_TO_REAL(Oee.RunMs) / UDINT_TO_REAL(denomA);
ELSE
    Oee.Availability := 0.0;
END_IF
Oee.PerfValid := (Oee.IdealCycleMs > 0) AND (Oee.RunMs > 0);
IF Oee.PerfValid THEN
    Oee.Performance := UDINT_TO_REAL(Oee.IdealCycleMs) * UDINT_TO_REAL(GoodCount + NokCount)
                       / UDINT_TO_REAL(Oee.RunMs);
    IF Oee.Performance > 1.0 THEN
        Oee.Performance := 1.0;          // faster than ideal caps at 100% (standard practice)
    END_IF
ELSE
    Oee.Performance := 0.0;
END_IF
total := GoodCount + NokCount;
Oee.QualValid := total > 0;
IF Oee.QualValid THEN
    Oee.Quality := UDINT_TO_REAL(GoodCount) / UDINT_TO_REAL(total);
ELSE
    Oee.Quality := 0.0;
END_IF
// product of VALID factors only; OEE valid iff at least one factor is valid
Oee.Oee := 1.0;
Oee.OeeValid := FALSE;
IF Oee.AvailValid THEN Oee.Oee := Oee.Oee * Oee.Availability; Oee.OeeValid := TRUE; END_IF
IF Oee.PerfValid  THEN Oee.Oee := Oee.Oee * Oee.Performance;  Oee.OeeValid := TRUE; END_IF
IF Oee.QualValid  THEN Oee.Oee := Oee.Oee * Oee.Quality;      Oee.OeeValid := TRUE; END_IF
IF NOT Oee.OeeValid THEN
    Oee.Oee := 0.0;
END_IF
END_METHOD

// §8.5.1 — attribute elapsed time to run/down/idle, recompute factors, sample ring.
METHOD PROTECTED _M_OeeUpdate
VAR
    currentTime : TIME;
    deltaMs     : UDINT;
END_VAR
currentTime := TIME();                 // monotonic duration clock
IF _oeeLast = T#0S THEN
    _oeeLast := currentTime;
    RETURN;
END_IF
deltaMs := TIME_TO_UDINT(currentTime) - TIME_TO_UDINT(_oeeLast); // wrap-safe on UDINT subtraction
_oeeLast := currentTime;
IF _exec = E_ExecState.BUSY THEN
    Oee.RunMs := Oee.RunMs + deltaMs;
ELSIF (_exec = E_ExecState.ERROR) OR AlarmLog.Blocking THEN
    Oee.DownMs := Oee.DownMs + deltaMs;
ELSE
    Oee.IdleMs := Oee.IdleMs + deltaMs;
END_IF
_M_OeeCompute();
_oeeSampMs := _oeeSampMs + deltaMs;
IF _oeeSampMs >= PL_Fraktal.OEE_SAMPLE_MS THEN
    _oeeSampMs := 0;
    OeeTrendHead := (OeeTrendHead MOD PL_Fraktal.MAX_OEE_SAMPLES) + 1;
    OeeTrend[OeeTrendHead].Availability := Oee.Availability;
    OeeTrend[OeeTrendHead].Performance  := Oee.Performance;
    OeeTrend[OeeTrendHead].Quality      := Oee.Quality;
    OeeTrend[OeeTrendHead].Oee          := Oee.Oee;
    OeeTrend[OeeTrendHead].OeeValid     := Oee.OeeValid;
END_IF
END_METHOD

// §3.16.3 EVENT_PART_PROCESSING_ABORTED — the part leaves without a valid result
// (fault, abort, manual removal). Called automatically on Unit ERROR entry.
METHOD PROTECTED _M_PartAborted
IF (_carrier = 0) OR NOT Part.Present THEN
    RETURN;
END_IF
Part.Result.Verdict := E_Verdict.NONE;
IF (_exec = E_ExecState.ERROR) AND (Part.Result.ReasonCode = E_Reason.NONE) THEN
    Part.Result.ReasonCode := _diag.ReasonCode;
END_IF
_M_PartEvent(Reason := E_Reason.EVENT_PART_PROCESSING_ABORTED,
    Text := 'std.event.partAborted: ');
_M_HostEvent(Kind := E_HostEventKind.PROCESSING_ABORTED, PartUid := Part.Uid,
    Subject := '', Value := '',
    Verdict := E_Verdict.NONE, ReasonCode := Part.Result.ReasonCode);
Part.Present := FALSE;
END_METHOD

// §3.16.3 — one canonical part-lifecycle event: instant come+gone MESSAGE ring entry.
METHOD PRIVATE _M_PartEvent
VAR_INPUT
    Reason : E_Reason;
    Text : STRING(255);
END_VAR
VAR
    slot : INT;
    txt : STRING(255);
END_VAR
txt := CONCAT(Text, Part.Uid);
slot := AlarmLog.Raise(Reason := Reason, Text := txt, Source := _name,
    Severity := E_Severity.LOW, Category := E_Category.PROCESS,
    ResetClass := E_ResetClass.AUTO_RESET);
IF slot > 0 THEN
    AlarmLog.Gone(Slot := slot);
END_IF
END_METHOD

// §3.16.3 EVENT_PART_PROCESSED — stamp the verdict, write the carrier FIRST
// (result-before-event contract), then raise the event. The Uid and result stay
// published until the next part so the HMI shows the last outcome.
METHOD PROTECTED _M_PartProcessed : BOOL
VAR_INPUT
    Verdict : E_Verdict;
    Reason : E_Reason;
END_VAR
_M_PartProcessed := FALSE;
IF (_carrier = 0) OR NOT Part.Present THEN
    RETURN;
END_IF
// A reject without a first-out reason cannot satisfy the KPI or host contract.
// Reject it before writing the carrier so result-before-event remains atomic.
IF (Verdict = E_Verdict.NOK) AND (Reason = E_Reason.NONE) THEN
    _M_Fault(E_Reason.RESULT_RECORD_REJECTED, 'std.error.nokReasonRequired');
    RETURN;
END_IF
Part.Result.Verdict := Verdict;
Part.Result.ReasonCode := Reason;
Part.Result.StationPath := _name;
Part.Result.Stamp := F_Now();
Part.Result.TimeSynchronized := F_TimeSynchronized();
IF NOT _carrier.WriteResult(Ctx := Part) THEN
    _M_Fault(E_Reason.CARRIER_WRITE_FAILED, 'std.error.partCarrierWriteFailed');
    RETURN;
END_IF
// §8.11.2 — counters increment HERE, from the verdict; an NOK carries its
// first-out ReasonCode so scrap is analysable by cause (§8.8 vocabulary).
CASE Verdict OF
    E_Verdict.OK:     CountGood();
    E_Verdict.NOK:
        IF NOT CountNok(Reason := Reason) THEN
            RETURN;
        END_IF
    E_Verdict.REWORK: CountRework();
ELSE
    ;                                // NONE: no count — the part left unjudged
END_CASE
_M_PartEvent(Reason := E_Reason.EVENT_PART_PROCESSED, Text := 'std.event.partProcessed: ');
_M_HostEvent(Kind := E_HostEventKind.PROCESSED, PartUid := Part.Uid,
    Subject := '', Value := '',
    Verdict := Verdict, ReasonCode := Reason);
Part.Present := FALSE;
_M_PartProcessed := TRUE;
END_METHOD

// §3.16.3 EVENT_PART_RECEIVED — confirm identity at station entry via the carrier.
// FALSE with a CARRIER_READ_FAILED fault on a failed read (never silent), FALSE
// silently when no carrier is configured (§3.9 feature selectability).
METHOD PROTECTED _M_PartReceived : BOOL
VAR
    i : INT;
END_VAR
_M_PartReceived := FALSE;
IF _carrier = 0 THEN
    RETURN;
END_IF
Part.Uid := '';                              // station entry = fresh identity read
IF NOT _carrier.ReadContext(Ctx := Part) THEN
    _M_Fault(E_Reason.CARRIER_READ_FAILED, 'std.error.partCarrierReadFailed');
    RETURN;
END_IF
Part.Result.Verdict := E_Verdict.NONE;       // this station's outcome starts empty
Part.Result.ReasonCode := E_Reason.NONE;
Part.Result.StationPath := _name;
FOR i := 1 TO PL_Fraktal.MAX_RESULTS DO
    Part.Result.Records[i].Name := '';
END_FOR
_M_PartEvent(Reason := E_Reason.EVENT_PART_RECEIVED, Text := 'std.event.partReceived: ');
_M_HostEvent(Kind := E_HostEventKind.PART_RECEIVED, PartUid := Part.Uid,
    Subject := '', Value := '',
    Verdict := E_Verdict.NONE, ReasonCode := E_Reason.NONE);
_M_PartReceived := TRUE;
END_METHOD

// §3.16.1 — append one measured value to this part's result (test cells).
// FALSE when the bounded record table is full (RESULT_RECORD_REJECTED semantics).
METHOD PROTECTED _M_PartRecord : BOOL
VAR_INPUT
    RecordName : STRING(64);
    Value : LREAL;
    Minimum : LREAL;
    Maximum : LREAL;
    Target : LREAL;
    EngUnit : STRING(16);
END_VAR
VAR
    i : INT;
END_VAR
_M_PartRecord := FALSE;
IF NOT Part.Present THEN
    RETURN;
END_IF
FOR i := 1 TO PL_Fraktal.MAX_RESULTS DO
    IF Part.Result.Records[i].Name = '' THEN
        Part.Result.Records[i].Name := RecordName;
        Part.Result.Records[i].Value := Value;
        Part.Result.Records[i].Minimum := Minimum;
        Part.Result.Records[i].Maximum := Maximum;
        Part.Result.Records[i].Target := Target;
        Part.Result.Records[i].Unit := EngUnit;
        Part.Result.Records[i].InTol := (Maximum <= Minimum)
            OR ((Value >= Minimum) AND (Value <= Maximum));
        _M_PartRecord := TRUE;
        RETURN;
    END_IF
END_FOR
END_METHOD

// §3.16.3 EVENT_PART_PROCESSING_STARTED — the value-adding sequence begins.
METHOD PROTECTED _M_PartStarted
IF (_carrier = 0) OR NOT Part.Present THEN
    RETURN;
END_IF
_M_PartEvent(Reason := E_Reason.EVENT_PART_PROCESSING_STARTED,
    Text := 'std.event.partProcessingStarted: ');
_M_HostEvent(Kind := E_HostEventKind.PROCESSING_STARTED, PartUid := Part.Uid,
    Subject := '', Value := '',
    Verdict := E_Verdict.NONE, ReasonCode := E_Reason.NONE);
END_METHOD

// §6.9/§3.10(a') — overlay the pending stall after the common mirror refresh.
METHOD PROTECTED _M_PublishStatus
SUPER^._M_PublishStatus();
// §8.11.4(f)/§8.11.3 — one declaration, two views. Derived AFTER dispatch so the
// wait class reflects the step record this scan just set, not the previous one.
// §3.13 — live row state for the flow chart: how long the active step has run,
// and whether it outran its declared guard (the same watchdog §6.9 stalls on).
IF _exec = E_ExecState.BUSY THEN
    CurrentStepElapsed := DWORD_TO_TIME(TIME_TO_DWORD(TIME()) - _stepSinceMs);
ELSE
    CurrentStepElapsed := T#0S;
END_IF
CurrentStepTimedOut := _tStall.Q;
Starved := (_exec = E_ExecState.BUSY) AND (CurrentStep.TimeClass = E_TimeClass.WAIT_UPSTREAM);
Blocked := (_exec = E_ExecState.BUSY) AND (CurrentStep.TimeClass = E_TimeClass.WAIT_DOWNSTREAM);
// §8.11.3 — classify into the fixed machine-state set (priority: fault first,
// then planned states, then line attribution, then producing/idle).
IF (_exec = E_ExecState.ERROR) OR AlarmLog.Blocking THEN
    MachineState := E_MachineState.DOWN;
ELSIF _mode = E_Mode.CHANGEOVER THEN
    MachineState := E_MachineState.CHANGEOVER;
ELSIF Blocked THEN
    MachineState := E_MachineState.BLOCKED;
ELSIF Starved THEN
    MachineState := E_MachineState.STARVED;
ELSIF _exec = E_ExecState.BUSY THEN
    MachineState := E_MachineState.PRODUCING;
ELSIF _stopReq OR (_exec = E_ExecState.ABORTED) THEN
    MachineState := E_MachineState.STOPPED;
ELSE
    MachineState := E_MachineState.IDLE;
END_IF
Status.ControlDomainId := ControlDomain.Id;
Domain := ControlDomain;
Safety := ControlDomain.Safety;             // read-only HMI mirror; ownership stays in domain
ControlPower := ControlDomain.ControlPower;
IF (_exec <> E_ExecState.ERROR) AND (Pending.ReasonCode <> E_Reason.NONE) THEN
    Status.Diagnostic := Pending;
END_IF
END_METHOD

// §6.9(a) — fixed ring, newest at HistoryHead; never allocates
METHOD PROTECTED _M_PushHistory
VAR_INPUT
    D : ST_Diagnostic;
END_VAR
HistoryHead := (HistoryHead MOD PL_Fraktal.MAX_DIAG_RING) + 1;
History[HistoryHead] := D;
END_METHOD

// §8.11.4(d)/§8.12 — a Low-severity maintenance event: informs planning, does not
// stop the cycle. Instant come+gone ring entry (the trend data lives in Profiler).
METHOD PROTECTED _M_RaiseMaintenance
VAR_INPUT
    Reason : E_Reason;
    Text : STRING(255);
END_VAR
VAR
    slot : INT;
END_VAR
slot := AlarmLog.Raise(Reason := Reason, Text := Text, Source := _name,
    Severity := E_Severity.LOW, Category := E_Category.SYSTEM,
    ResetClass := E_ResetClass.AUTO_RESET);
IF slot > 0 THEN
    AlarmLog.Gone(Slot := slot);
END_IF
END_METHOD

// §3.8b — route a published editable field to the module that registered it.
// WriteConfig already owns access and root-path checks; the recursive walk finds
// the owner by Scope, and that module rechecks revision, type, range, domain and
// its own invariants before storing. A type whose values are declared through
// M_RegisterConfig* therefore needs no override at all, which is the point: a new
// module type costs no routing code (§1.1 O1). Framework-owned keys never reach
// here — _M_WriteBaseConfig answers those first. An override that adds
// hand-written routing shall call SUPER^ first and keep its own answer only when
// the base declines.
METHOD PROTECTED _M_RouteConfigWrite : BOOL
VAR_INPUT
    TargetPath : STRING(255);
    WriteKey   : STRING(160);
    Revision   : UDINT;
    TextValue  : STRING(255);
END_VAR
// RequiresReady is a question about THIS root's state, which the owning child
// cannot see from where it sits, so the root answers it on the way down.
_M_RouteConfigWrite := M_ApplyConfigWrite(Scope := TargetPath,
    WriteKey := WriteKey, Revision := Revision, TextValue := TextValue,
    // Another model's record is not what the machine is running on.
    RootReady := (_exec = E_ExecState.READY) OR (_pModelView <> 0));
END_METHOD

// Framework-owned typed handlers. Stable keys are independent of browse paths;
// capability revision 1 accepts exact enum ordinals and only while READY.
//
// Commit := FALSE validates and stores nothing — the staging pass of a §3.8b set
// load. The root's own ModePolicy keys are published as STATION_CFG
// capabilities, so they are in every station set and have to stage through the
// same validator that writes them, for the same reason every module's do.
METHOD PRIVATE _M_WriteBaseConfig : BOOL
VAR_INPUT
    TargetPath : STRING(255);
    WriteKey   : STRING(160);
    Revision   : UDINT;
    TextValue  : STRING(255);
    Commit     : BOOL;
END_VAR
VAR
    i      : INT;
    key    : STRING(160);
    shield : E_ModeSwitchShield;
    style  : E_ModeSwitchStyle;
END_VAR
_M_WriteBaseConfig := FALSE;
IF (TargetPath <> Status.Name) OR (Revision <> 1) OR (_exec <> E_ExecState.READY) THEN
    RETURN;
END_IF
FOR i := 0 TO PL_Fraktal.MODE_COUNT - 1 DO
    key := CONCAT('unit.modePolicy.', CONCAT(TO_STRING(i), '.shield'));
    IF WriteKey = key THEN
        IF TextValue = '0' THEN
            shield := E_ModeSwitchShield.INTERRUPTIBLE;
        ELSIF TextValue = '1' THEN
            shield := E_ModeSwitchShield.CONFIRM;
        ELSIF TextValue = '2' THEN
            shield := E_ModeSwitchShield.BLOCKED_WHILE_RUNNING;
        ELSE
            RETURN;
        END_IF
        IF Commit THEN
            ModePolicy[i].Shield := shield;
            _modePolicyStored[i].Shield := shield;
        END_IF
        _M_WriteBaseConfig := TRUE;
        RETURN;
    END_IF
    key := CONCAT('unit.modePolicy.', CONCAT(TO_STRING(i), '.style'));
    IF WriteKey = key THEN
        IF TextValue = '0' THEN
            style := E_ModeSwitchStyle.GRACEFUL;
        ELSIF TextValue = '1' THEN
            style := E_ModeSwitchStyle.IMMEDIATE;
        ELSE
            RETURN;
        END_IF
        IF Commit THEN
            ModePolicy[i].Style := style;
            _modePolicyStored[i].Style := style;
        END_IF
        _M_WriteBaseConfig := TRUE;
        RETURN;
    END_IF
END_FOR
END_METHOD

// Application override resolves ChannelPath in THIS root's approved I/O catalog,
// refuses input/safety/unmapped channels, applies its channel-specific §7.6 permit,
// and routes only an approved mapped output. ForceChannel already owns MANUAL,
// stopped/READY, access and audit. Base fails closed.
METHOD PROTECTED _M_RouteForceChannel : BOOL
VAR_INPUT
    ChannelPath : STRING(255);
    Force       : BOOL;
    BoolText    : STRING(255);
    AnalogText  : STRING(160);
END_VAR
_M_RouteForceChannel := FALSE;
END_METHOD

// §7.6.1 — route a manual command to the module that owns TargetPath, through
// the SAME registered-child walk that already carries configuration writes.
//
// This used to return FALSE and leave every Unit to hand-write its own routing
// chain. That is a call a project must remember for correctness (§1.1 O1), and
// it failed exactly as O1 predicts: the press registered eight children and
// routed three, so five modules published manual commands the HMI rendered and
// the Unit silently refused. A registered child is now commandable BECAUSE it
// is registered.
//
// An override still wins, so a Unit with genuinely special routing keeps it;
// it should call SUPER^ first and keep its own answer only when the base
// declines.
METHOD PROTECTED _M_RouteManual : BOOL
VAR_INPUT
    TargetPath : STRING(255);
    Value : DINT;
END_VAR
_M_RouteManual := M_ApplyManual(Scope := TargetPath, Value := Value);
END_METHOD

// §3.13 — keep the published flow chart in step with the chain.
// Called only from _M_SetStep, so every step of every chain lands here exactly
// once per visit and a chain author writes nothing (§1.1 O1). Rows are matched by
// StepNo, appended on first sight and bounded: an overflowing chain publishes the
// first MAX_SEQUENCE_STEPS rows rather than dropping the chart.
METHOD PROTECTED _M_RecordSequenceStep
VAR_INPUT
    StepNo        : INT;
    StepName      : STRING(120);
    Awaits        : I_Module;
    AwaitingLabel : STRING(120);
    TimeClass     : E_TimeClass;
    ExpectedTime  : TIME;
    Branch        : INT;           // §6.12 concurrent leg, 0 = the chain's main line
END_VAR
VAR
    i    : INT;
    hit  : INT;
    path : STRING(255);
END_VAR
hit := 0;
FOR i := 1 TO SequenceStepCount DO
    IF SequenceStepDef[i].StepNo = StepNo THEN
        hit := i;
        EXIT;
    END_IF
END_FOR
IF hit = 0 THEN
    IF SequenceStepCount >= PL_Fraktal.MAX_SEQUENCE_STEPS THEN
        RETURN;                        // bounded: publish what fits, never overrun
    END_IF
    SequenceStepCount := SequenceStepCount + 1;
    hit := SequenceStepCount;
    // §3.10.2 — the static half of this row (StepNo, StepName, the awaited path)
    // is served through the manifest, NOT cyclically, and the HMI refetches only
    // when ConfigRev changes. Rows are discovered by visit, so a chart that grows
    // after the HMI's fetch would render every new row with StepNo 0 and no text.
    // Only the append marks it: a re-visit rewrites identical values.
    //
    // MARKED, not bumped: the revision is raised once the chart stops growing
    // (_M_ChartRevCyclic). Invalidating the whole manifest per discovered row
    // made entering a 15-step mode cost fifteen full refetches.
    _chartDirty := TRUE;
    _chartTouchedMs := TIME_TO_DWORD(TIME());
END_IF
// The drill-down target is the module the step DECLARES it commands. Reading it
// here is what makes the link unambiguous: no IF/CASE chose it (§3.13).
path := '';
IF Awaits <> 0 THEN
    path := Awaits.Name;
END_IF
// Static half: fixed from this first visit, published through the manifest.
SequenceStepDef[hit].StepNo        := StepNo;
SequenceStepDef[hit].Branch        := Branch;
SequenceStepDef[hit].TimeClass     := TimeClass;
SequenceStepDef[hit].ExpectedTime  := ExpectedTime;
SequenceStepDef[hit].StepName      := StepName;
SequenceStepDef[hit].AwaitingLabel := AwaitingLabel;
SequenceStepDef[hit].AwaitsPath    := path;
SequenceSteps[hit].Visited := TRUE;
// §6.12 — the LEG owns the clock, because a leg runs exactly one step at a time.
// A different row on this leg means the step just changed.
IF ActiveSteps[Branch].RowIdx <> hit THEN
    SequenceSteps[hit].WarningActive := FALSE;   // §6.9(e) this visit starts clean
    _M_SequenceAnnotationClear(RowIdx := hit, IsError := FALSE);
    _branchSinceMs[Branch] := TIME_TO_DWORD(TIME());
    ActiveSteps[Branch].RowIdx := hit;
    ActiveSteps[Branch].Elapsed := T#0S;
    ActiveSteps[Branch].TimedOut := FALSE;
    IF Branch = 0 THEN
        _stepSinceMs := _branchSinceMs[0];
        CurrentStepElapsed := T#0S;
    END_IF
END_IF
_branchTouched[Branch] := TRUE;
ActiveSteps[Branch].Elapsed :=
    DWORD_TO_TIME(TIME_TO_DWORD(TIME()) - _branchSinceMs[Branch]);
// A leg carries its own guard: the §6.9 stall watchdog is singular and follows the
// main line, so without this a leg could overrun for ever with nothing to show.
ActiveSteps[Branch].TimedOut := (ExpectedTime > T#0S)
    AND (ActiveSteps[Branch].Elapsed > ExpectedTime);
// The row recorded last IS the step action executing right now, which is what makes
// it the correct target for a §6.9 raise or a §6.9(e) message raised further down
// that same action - on the main line or on any leg.
_seqIndex := hit;
END_METHOD

// §3.13 — drop the published flow chart so the next mode builds its own.
//
// The row table is DISCOVERED by visit (§6.5), which is what makes it free to
// author - but discovery has no end: without this the table becomes the union of
// every chain run since boot. After AUTO then HOME the operator would be shown
// AUTO's rows and HOME's together with only some of them live, and the union of
// the press demo's three modes is 29 rows against a bound of 32. A mode is the
// natural boundary: within one mode a re-run keeps its rows, so Visited and
// LastDuration stay meaningful across cycles.
//
// Bounded by the count actually in use, not by MAX_SEQUENCE_STEPS: clearing rows
// nobody published would cost the whole table on every mode change (§1.1 O10 -
// deterministic scan time).
METHOD PROTECTED _M_ResetSequenceRows
VAR
    i : INT;
    e : ST_SequenceStep;
    x : ST_SequenceStepDef;
    c : ST_SequenceCursor;
    a : ST_SequenceAnnotation;
END_VAR
IF SequenceStepCount > 0 THEN
    // §3.10.2 — the rows this clears are published through the manifest, so the
    // HMI's cached copy is now describing a chart that no longer exists. Guarded
    // by the count: a mode change with nothing published changed no manifest and
    // must not cost a refetch.
    //
    // Marked rather than bumped, and for the same reason as the append: the
    // clear and the regrow that follows it are ONE episode, so they should cost
    // one refetch between them, not one plus one per rediscovered row.
    _chartDirty := TRUE;
    _chartTouchedMs := TIME_TO_DWORD(TIME());
END_IF
FOR i := 1 TO SequenceStepCount DO
    SequenceSteps[i] := e;             // zero-initialized local: clears every field
    SequenceStepDef[i] := x;
END_FOR
SequenceStepCount := 0;
FOR i := 0 TO PL_Fraktal.MAX_PARALLEL_BRANCHES DO
    ActiveSteps[i] := c;
    _branchTouched[i] := FALSE;
END_FOR
FOR i := 1 TO SequenceAnnotationCount DO
    SequenceAnnotations[i] := a;
END_FOR
SequenceAnnotationCount := 0;
_seqIndex := 0;                        // nothing to stamp until the new chain steps
CurrentStepElapsed := T#0S;
END_METHOD

// §6.9 — attach an error or a message to a flow-chart row.
//
// One slot per (row, kind): re-annotating the same row with the same kind
// overwrites rather than accumulating, which is what makes it safe for the
// per-visit message latch to call this without tracking slots.
//
// Returns FALSE when the table is full. The CALLER has already set the row flag
// by then, deliberately: a full table costs the text, never the mark, so the
// chart still shows that something happened here (§5.6 degrade, never mislead).
METHOD PROTECTED _M_SequenceAnnotate : BOOL
VAR_INPUT
    RowIdx     : INT;
    IsError    : BOOL;
    Key        : STRING(120);
    SourcePath : STRING(80);
END_VAR
VAR
    i    : INT;
    slot : INT;
END_VAR
_M_SequenceAnnotate := FALSE;
IF (RowIdx < 1) OR (RowIdx > SequenceStepCount) THEN
    RETURN;
END_IF
slot := 0;
FOR i := 1 TO SequenceAnnotationCount DO
    IF (SequenceAnnotations[i].RowIdx = RowIdx)
    AND (SequenceAnnotations[i].IsError = IsError) THEN
        slot := i;
        EXIT;
    END_IF
END_FOR
IF slot = 0 THEN
    FOR i := 1 TO SequenceAnnotationCount DO
        IF SequenceAnnotations[i].RowIdx = 0 THEN     // freed by a clear
            slot := i;
            EXIT;
        END_IF
    END_FOR
END_IF
IF slot = 0 THEN
    IF SequenceAnnotationCount >= PL_Fraktal.MAX_SEQUENCE_ANNOTATIONS THEN
        RETURN;                                       // full: the mark stands, the text does not
    END_IF
    SequenceAnnotationCount := SequenceAnnotationCount + 1;
    slot := SequenceAnnotationCount;
END_IF
SequenceAnnotations[slot].RowIdx     := RowIdx;
SequenceAnnotations[slot].IsError    := IsError;
SequenceAnnotations[slot].Key        := Key;
SequenceAnnotations[slot].SourcePath := SourcePath;
_M_SequenceAnnotate := TRUE;
END_METHOD

// §6.9 — release annotations. RowIdx 0 means "every row" (the ERROR-cleared edge
// drops all error notes at once); otherwise just that row's note of that kind.
// Freed slots are reused before the table grows, so a chain that warns on many
// steps over many cycles does not exhaust it.
METHOD PROTECTED _M_SequenceAnnotationClear
VAR_INPUT
    RowIdx  : INT;
    IsError : BOOL;
END_VAR
VAR
    i : INT;
    e : ST_SequenceAnnotation;
END_VAR
FOR i := 1 TO SequenceAnnotationCount DO
    IF (SequenceAnnotations[i].IsError = IsError)
    AND ((RowIdx = 0) OR (SequenceAnnotations[i].RowIdx = RowIdx)) THEN
        SequenceAnnotations[i] := e;                  // RowIdx 0 marks the slot free
    END_IF
END_FOR
END_METHOD

// §6.5 — the ONE line per step: record for the §6.9 walk AND the §8.11.4 profiler
METHOD PROTECTED _M_SetStep
VAR_INPUT
    StepNo        : INT;
    StepName      : STRING(120);
    Awaits        : I_Module;
    AwaitingLabel : STRING(120);
    TimeClass     : E_TimeClass;
    ExpectedTime  : TIME;
END_VAR
VAR
    i : INT;
    e : ST_CondRecord;
END_VAR
IF StepNo <> CurrentStep.StepNo THEN
    _tStall(IN := FALSE);
    _M_ClearPending();
    FOR i := 1 TO PL_Fraktal.MAX_STEP_CONDS DO
        CurrentStep.Conds[i] := e;
    END_FOR
END_IF
CurrentStep.StepNo        := StepNo;
CurrentStep.StepName      := StepName;
CurrentStep.AwaitingLabel := AwaitingLabel;
CurrentStep.TimeClass     := TimeClass;
CurrentStep.ExpectedTime  := ExpectedTime;
_awaits := Awaits;
_M_RecordSequenceStep(StepNo := StepNo, StepName := StepName, Awaits := Awaits,
    AwaitingLabel := AwaitingLabel, TimeClass := TimeClass, ExpectedTime := ExpectedTime,
    Branch := 0);
Profiler.StepChanged(StepNo := StepNo, StepName := StepName, TimeClass := TimeClass,
    Expected := ExpectedTime);
END_METHOD

// §6.9 — build the pending stall reason: step -> awaited command -> first FALSE condition
METHOD PROTECTED _M_StallWalk
IF Pending.ReasonCode = E_Reason.NONE THEN
    Pending.Since := F_Now();
    Pending.TimeSynchronized := F_TimeSynchronized();
END_IF
Pending.ReasonCode := E_Reason.STEP_STALLED;
Pending.Severity   := E_Severity.LOW;
Pending.Category   := E_Category.PROCESS;
Pending.SourcePath := _name;
Pending.Description := 'std.diagnostic.stepStalled';
END_METHOD

// §3.4.2 — the sequence author calls this at each step boundary; returns TRUE when
// the sequence may advance. Steppable (default TRUE) is the PER-STEP stop-point flag:
// a step with Steppable := FALSE runs straight through even in SINGLE_STEP/HOLD_TO_RUN
// (group several motions into one operator step, or a step unsafe to pause mid-way).
// CONTINUOUS: always TRUE. SINGLE_STEP: TRUE once per StepRequest edge (only if
// Steppable). HOLD_TO_RUN: TRUE while held (only if Steppable). Interlocks are
// enforced by the modules regardless (this only paces the sequence).
METHOD PROTECTED _M_StepGate : BOOL
VAR_INPUT
    Steppable : BOOL;
END_VAR
IF NOT Steppable THEN
    _M_StepGate := TRUE;               // not a stop point: advance regardless of run style
    RETURN;
END_IF
CASE RunStyle OF
    E_RunStyle.SINGLE_STEP:
        _stepArm(CLK := _stepReq);
        _stepReq := FALSE;
        _M_StepGate := _stepArm.Q;      // one advance per request edge
    E_RunStyle.HOLD_TO_RUN:
        _M_StepGate := _holdRun;        // advance only while held (NON-SAFETY)
ELSE
    _M_StepGate := TRUE;                // CONTINUOUS
END_CASE
END_METHOD

// §3.4 — override to declare the type's mode set (baseline: AUTO + MANUAL)
METHOD PROTECTED _M_Supports : BOOL
VAR_INPUT
    Mode : E_Mode;
END_VAR
_M_Supports := (Mode = E_Mode.AUTO) OR (Mode = E_Mode.MANUAL);
END_METHOD

// §3.4.2 — a concrete Unit overrides to opt a mode into SINGLE_STEP/HOLD_TO_RUN.
// Base: only CONTINUOUS.
METHOD PROTECTED _M_SupportsRunStyle : BOOL
VAR_INPUT
    Style : E_RunStyle;
END_VAR
_M_SupportsRunStyle := (Style = E_RunStyle.CONTINUOUS);
END_METHOD

// §6.11 — returns the chosen option once and clears the request (0 = none yet)
METHOD PROTECTED _M_TakeDecision : INT
IF DecisionAnswer > 0 THEN
    _M_TakeDecision := DecisionAnswer;
    IF NOT _decisionResolutionLogged THEN
        _M_LogDecision(EventKey := 'std.audit.decisionOperatorResolved',
            SourcePath := Decision.SourcePath, Option := DecisionAnswer);
    END_IF
    _M_ClearDecisionState();
ELSE
    _M_TakeDecision := 0;
END_IF
END_METHOD

// §8.11 — called by the chain/verdict glue at part completion
METHOD CountGood : BOOL
GoodCount := GoodCount + 1;
CountGood := TRUE;
END_METHOD

// Sections 8.11.2 and 11.6: one authoritative NOK outcome path.
// Part.Uid is empty when the optional traceability carrier is not configured.
METHOD CountNok : BOOL
VAR_INPUT
    Reason : E_Reason;
END_VAR
CountNok := FALSE;
IF Reason = E_Reason.NONE THEN
    _M_Fault(E_Reason.RESULT_RECORD_REJECTED, 'std.error.nokReasonRequired');
    RETURN;
END_IF
IF NOT _M_HostEvent(Kind := E_HostEventKind.NOK, PartUid := Part.Uid,
        Subject := '', Value := '', Verdict := E_Verdict.NOK,
        ReasonCode := Reason) THEN
    _M_Fault(E_Reason.RESULT_RECORD_REJECTED, 'std.error.hostEventRejected');
    RETURN;
END_IF
NokCount := NokCount + 1;
NokReason := Reason;
CountNok := TRUE;
END_METHOD

// §8.11.2 — REWORK verdict counter (see CountGood)
METHOD CountRework : BOOL
ReworkCount := ReworkCount + 1;
CountRework := TRUE;
END_METHOD

// §3.10.2 — Unit facets after the composite walk (own catalog + children):
// model catalog and per-mode switch policy, both static between config edits.
METHOD M_AppendConfig : BOOL
VAR_INPUT
    Pager : REFERENCE TO FB_ConfigPager;
END_VAR
VAR
    i        : INT;
    metaIndex: INT;
    item     : STRING(255);
    writeKey : STRING(160);
    labelKey : STRING(160);  // std.config.modePolicy.<mode ordinal>.<shield|style>
    meta     : ST_AlarmMeta;
    seqIdx   : INT;
    seqBase  : STRING(255);
END_VAR
M_AppendConfig := SUPER^.M_AppendConfig(Pager := Pager);
IF _pLine <> 0 THEN
    _pLine^.M_AppendLineConfig(Pager := Pager, Scope := Status.Name);   // §3.8e
END_IF
Pager.M_AppendNumber(Scope := Status.Name, Item := 'StallTime',
    Number := TIME_TO_DINT(StallTime));
Pager.M_AppendNumber(Scope := Status.Name, Item := 'AvailableModelCount',
    Number := TO_DINT(AvailableModelCount));
FOR i := 1 TO AvailableModelCount DO
    item := CONCAT('AvailableModels/AvailableModels[',
        CONCAT(TO_STRING(i), ']/ModelCode'));
    Pager.M_Append(Scope := Status.Name, Item := item,
        ValueText := AvailableModels[i].ModelCode);
END_FOR
FOR i := 0 TO PL_Fraktal.MODE_COUNT - 1 DO
    item := CONCAT('ModePolicy/ModePolicy[', CONCAT(TO_STRING(i), ']/Shield'));
    writeKey := CONCAT('unit.modePolicy.', CONCAT(TO_STRING(i), '.shield'));
    labelKey := CONCAT('std.config.modePolicy.', CONCAT(TO_STRING(i), '.shield'));
    Pager.M_AppendCapability(Scope := Status.Name, Item := item,
        ValueText := TO_STRING(TO_DINT(ModePolicy[i].Shield)), WriteKey := writeKey,
        WriteRevision := 1, ConfigKind := E_ConfigKind.STATION_CFG,
        ValueType := E_ConfigValueType.NUMBER, Writable := TRUE,
        RequiresReady := TRUE, HasMinimum := TRUE, HasMaximum := TRUE,
        Minimum := 0.0, Maximum := 2.0, Unit := E_EngUnit.NONE, LabelKey := labelKey,
        EnumDomain := '0|1|2', EnumLabelKey := 'std.enum.modeSwitchShield',
        ClassId := '', MinReadLevel := E_AccessLevel.NONE,
        MinWriteLevel := E_AccessLevel.NONE, ModelScoped := FALSE);
    item := CONCAT('ModePolicy/ModePolicy[', CONCAT(TO_STRING(i), ']/Style'));
    writeKey := CONCAT('unit.modePolicy.', CONCAT(TO_STRING(i), '.style'));
    labelKey := CONCAT('std.config.modePolicy.', CONCAT(TO_STRING(i), '.style'));
    Pager.M_AppendCapability(Scope := Status.Name, Item := item,
        ValueText := TO_STRING(TO_DINT(ModePolicy[i].Style)), WriteKey := writeKey,
        WriteRevision := 1, ConfigKind := E_ConfigKind.STATION_CFG,
        ValueType := E_ConfigValueType.NUMBER, Writable := TRUE,
        RequiresReady := TRUE, HasMinimum := TRUE, HasMaximum := TRUE,
        Minimum := 0.0, Maximum := 1.0, Unit := E_EngUnit.NONE, LabelKey := labelKey,
        EnumDomain := '0|1', EnumLabelKey := 'std.enum.modeSwitchStyle',
        ClassId := '', MinReadLevel := E_AccessLevel.NONE,
        MinWriteLevel := E_AccessLevel.NONE, ModelScoped := FALSE);
END_FOR
Pager.M_AppendNumber(Scope := Status.Name, Item := 'AlarmLog/MetaCount',
    Number := TO_DINT(PL_ReasonCatalog.COUNT + AlarmLog.MetaCount));
// §8.8/§8.9: the standard catalog is generated from the numeric sources plus
// one symbol-keyed rationalization registry. Static metadata stays manifest-only.
FOR i := 1 TO PL_ReasonCatalog.COUNT DO
    IF NOT F_ReasonMetaByIndex(Index := i, Meta := meta) THEN
        EXIT;
    END_IF
    item := CONCAT('AlarmLog/Meta/Meta[', CONCAT(TO_STRING(i), ']/ReasonCode'));
    Pager.M_AppendNumber(Scope := Status.Name, Item := item,
        Number := TO_DINT(meta.ReasonCode));
    item := CONCAT('AlarmLog/Meta/Meta[', CONCAT(TO_STRING(i), ']/OperatorAction'));
    Pager.M_Append(Scope := Status.Name, Item := item,
        ValueText := meta.OperatorAction);
    item := CONCAT('AlarmLog/Meta/Meta[', CONCAT(TO_STRING(i), ']/Consequence'));
    Pager.M_Append(Scope := Status.Name, Item := item,
        ValueText := meta.Consequence);
    item := CONCAT('AlarmLog/Meta/Meta[', CONCAT(TO_STRING(i), ']/Priority'));
    Pager.M_AppendNumber(Scope := Status.Name, Item := item,
        Number := TO_DINT(meta.Priority));
    item := CONCAT('AlarmLog/Meta/Meta[', CONCAT(TO_STRING(i), ']/Category'));
    Pager.M_AppendNumber(Scope := Status.Name, Item := item,
        Number := TO_DINT(meta.Category));
    item := CONCAT('AlarmLog/Meta/Meta[', CONCAT(TO_STRING(i), ']/Shelvable'));
    IF meta.Shelvable THEN
        Pager.M_Append(Scope := Status.Name, Item := item, ValueText := 'TRUE');
    ELSE
        Pager.M_Append(Scope := Status.Name, Item := item, ValueText := 'FALSE');
    END_IF
END_FOR
// External/application libraries may append rationalized reasons not present in
// the shipped registry. RegisterMetaFull enforces their complete record.
FOR i := 1 TO AlarmLog.MetaCount DO
    metaIndex := PL_ReasonCatalog.COUNT + i;
    item := CONCAT('AlarmLog/Meta/Meta[', CONCAT(TO_STRING(metaIndex), ']/ReasonCode'));
    Pager.M_AppendNumber(Scope := Status.Name, Item := item,
        Number := TO_DINT(AlarmLog.Meta[i].ReasonCode));
    item := CONCAT('AlarmLog/Meta/Meta[', CONCAT(TO_STRING(metaIndex), ']/OperatorAction'));
    Pager.M_Append(Scope := Status.Name, Item := item,
        ValueText := AlarmLog.Meta[i].OperatorAction);
    item := CONCAT('AlarmLog/Meta/Meta[', CONCAT(TO_STRING(metaIndex), ']/Consequence'));
    Pager.M_Append(Scope := Status.Name, Item := item,
        ValueText := AlarmLog.Meta[i].Consequence);
    item := CONCAT('AlarmLog/Meta/Meta[', CONCAT(TO_STRING(metaIndex), ']/Priority'));
    Pager.M_AppendNumber(Scope := Status.Name, Item := item,
        Number := TO_DINT(AlarmLog.Meta[i].Priority));
    item := CONCAT('AlarmLog/Meta/Meta[', CONCAT(TO_STRING(metaIndex), ']/Category'));
    Pager.M_AppendNumber(Scope := Status.Name, Item := item,
        Number := TO_DINT(AlarmLog.Meta[i].Category));
    item := CONCAT('AlarmLog/Meta/Meta[', CONCAT(TO_STRING(metaIndex), ']/Shelvable'));
    IF AlarmLog.Meta[i].Shelvable THEN
        Pager.M_Append(Scope := Status.Name, Item := item, ValueText := 'TRUE');
    ELSE
        Pager.M_Append(Scope := Status.Name, Item := item, ValueText := 'FALSE');
    END_IF
END_FOR
// §3.13/§3.10.2 — the static definition of each flow-chart row. The Item fragment
// reproduces the browse path the LIVE half is published under, so the HMI mapper
// reads `SequenceSteps[i]/StepName` without knowing it arrived by a different
// route: one row structure, half of it live, half fetched once and cached.
// Bounded by the discovered count, so an empty chain appends nothing.
FOR seqIdx := 1 TO SequenceStepCount DO
    seqBase := CONCAT('SequenceSteps/SequenceSteps[', CONCAT(TO_STRING(seqIdx), ']/'));
    Pager.M_AppendNumber(Scope := Status.Name, Item := CONCAT(seqBase, 'StepNo'),
        Number := TO_DINT(SequenceStepDef[seqIdx].StepNo));
    Pager.M_AppendNumber(Scope := Status.Name, Item := CONCAT(seqBase, 'Branch'),
        Number := TO_DINT(SequenceStepDef[seqIdx].Branch));
    Pager.M_AppendNumber(Scope := Status.Name, Item := CONCAT(seqBase, 'TimeClass'),
        Number := TO_DINT(SequenceStepDef[seqIdx].TimeClass));
    Pager.M_AppendNumber(Scope := Status.Name, Item := CONCAT(seqBase, 'ExpectedTime'),
        Number := TIME_TO_DINT(SequenceStepDef[seqIdx].ExpectedTime));
    Pager.M_Append(Scope := Status.Name, Item := CONCAT(seqBase, 'StepName'),
        ValueText := SequenceStepDef[seqIdx].StepName);
    Pager.M_Append(Scope := Status.Name, Item := CONCAT(seqBase, 'AwaitingLabel'),
        ValueText := SequenceStepDef[seqIdx].AwaitingLabel);
    Pager.M_Append(Scope := Status.Name, Item := CONCAT(seqBase, 'AwaitsPath'),
        ValueText := SequenceStepDef[seqIdx].AwaitsPath);
END_FOR
END_METHOD

// §3.8b — inject this deployment's parameter-set store at Setup, the same shape
// as SetPartCarrier and the §3.8 recipe provider. Absent means save/load/list are
// not offered at all, published as StorePresent = FALSE — a stated fact rather
// than a request that fails the first time an operator tries it.
METHOD SetConfigStore : BOOL
VAR_INPUT
    Store : I_ConfigStore;
END_VAR
SetConfigStore := FALSE;
IF Store = 0 THEN
    RETURN;
END_IF
_configStore := Store;
ConfigPersist.StorePresent := TRUE;
ConfigPersist.StoreKind := Store.M_Kind();
SetConfigStore := TRUE;
END_METHOD

// §3.8b — substitute the durability provider. The shipped LOCAL_RETAIN writer is
// used when nothing is injected, so this exists for a deployment whose
// configuration genuinely lives somewhere else (a file, a database, an MES) —
// not as one more thing every station has to remember to wire (§1.1 O1).
METHOD SetConfigPersistence : BOOL
VAR_INPUT
    Provider : I_ConfigPersistence;
END_VAR
SetConfigPersistence := FALSE;
IF Provider = 0 THEN
    RETURN;
END_IF
_persistence := Provider;
SetConfigPersistence := TRUE;
END_METHOD

// §3.8b — declare how long an accepted write may take to become durable. The
// clause says "within a declared bounded window", and the point of DECLARING it
// is that different stores have honestly different latencies: a retentive write
// is milliseconds, an MES round trip is not. A deployment that leaves this alone
// gets PL_Fraktal.CONFIG_PERSIST_WINDOW_MS.
//
// Zero means "durable immediately or not at all", which is the correct
// declaration for a store that either completes in the same scan or has failed.
METHOD SetConfigPersistWindow : BOOL
VAR_INPUT
    WindowMs : UDINT;
END_VAR
ConfigPersist.WindowMs := WindowMs;
SetConfigPersistWindow := TRUE;
END_METHOD

// §3.8b — declare what this station DOES about a lost configuration image.
// DEFAULTS_AND_ANNUNCIATE is the shipped default; a station whose commissioned
// values are the difference between a good part and a wrecked tool declares
// BLOCK_UNTIL_ACKNOWLEDGED instead. It is a DEPLOYMENT decision on purpose: no
// module type is in a position to know which of the two its station is, which is
// why a module reporting a loss never decides the consequence of one.
METHOD SetConfigRestorePolicy : BOOL
VAR_INPUT
    Policy : E_ConfigRestorePolicy;
END_VAR
ConfigPersist.RestorePolicy := Policy;
SetConfigRestorePolicy := TRUE;
END_METHOD

// §3.8b — an accepted write is LIVE. This starts the clock on it becoming
// DURABLE, and the root publishes PersistPending until it is. Called from every
// path that accepts a value, so no project and no module type has to remember
// that a write it just made is not yet safe (§1.1 O1).
METHOD PROTECTED _M_MarkPersistPending
IF NOT ConfigPersist.Pending THEN
    ConfigPersist.Pending := TRUE;
    ConfigPersist.PendingSince := F_Now();
END_IF
// The window runs from the LATEST accepted write, because that is the one whose
// durability is in question; PendingSince stays at the start of the episode so
// an operator can see how long this station has been unsafe.
_persistSinceMs := TIME_TO_DWORD(TIME());
ConfigPersist.Failed := FALSE;
IF _persistEvt > 0 THEN
    AlarmLog.Gone(Slot := _persistEvt);
    _persistEvt := 0;
END_IF
IF _persistence = 0 THEN
    RETURN;                                // no provider: the window will expire
END_IF
IF NOT _persistence.M_Request() THEN
    _M_ConfigPersistFailed();              // refused before it began is a failure
END_IF
END_METHOD

// §3.8b — the store rejected the write, or the declared window elapsed with it
// still not durable. Pending stays TRUE because the value is STILL not durable;
// Failed says it will not get there on its own.
//
// Deliberately NOT retried in a loop: a store that cannot write is not fixed by
// asking again every scan, and a retry storm would bury the one annunciation an
// operator needs. The next accepted write re-arms it.
METHOD PRIVATE _M_ConfigPersistFailed
ConfigPersist.Failed := TRUE;
IF _persistEvt > 0 THEN
    RETURN;                                // one standing event, not one per scan
END_IF
// AUTO_RESET: loud enough to see, never blocking. A station whose configuration
// will not persist can still finish the parts already in it, and the operator is
// told BEFORE the restart that would otherwise reveal this silently.
_persistEvt := AlarmLog.Raise(Reason := E_Reason.CONFIG_PERSIST_FAILED,
    Text := 'std.error.configPersistFailed', Source := _name,
    Severity := E_Severity.MED, Category := E_Category.SYSTEM,
    ResetClass := E_ResetClass.AUTO_RESET);
END_METHOD

// §3.8b — drive the durability provider and hold the declared window to
// account. "Within a declared bounded window" is a promise, and a promise
// nobody measures is the hope the clause replaces: the window is checked here
// every scan, and exceeding it publishes PersistFailed.
METHOD PRIVATE _M_ConfigPersistCyclic
VAR
    busy    : BOOL;
    elapsed : DWORD;
END_VAR
busy := FALSE;
IF _persistence <> 0 THEN
    busy := _persistence.M_Cyclic();
END_IF
IF NOT ConfigPersist.Pending THEN
    RETURN;
END_IF
IF busy THEN
    // Unsigned subtraction, so the monotonic millisecond counter wrapping does
    // not fabricate an expired window (TC3 §8.11).
    elapsed := TIME_TO_DWORD(TIME()) - _persistSinceMs;
    IF elapsed > TO_DWORD(ConfigPersist.WindowMs) THEN
        _M_ConfigPersistFailed();
    END_IF
    RETURN;
END_IF
// Nothing in flight. Either it finished, or there is no provider to finish it.
IF _persistence = 0 THEN
    elapsed := TIME_TO_DWORD(TIME()) - _persistSinceMs;
    IF elapsed > TO_DWORD(ConfigPersist.WindowMs) THEN
        _M_ConfigPersistFailed();
    END_IF
    RETURN;
END_IF
IF _persistence.M_Failed() THEN
    _M_ConfigPersistFailed();
    RETURN;
END_IF
ConfigPersist.Pending := FALSE;
ConfigPersist.Failed := FALSE;
IF _persistEvt > 0 THEN
    AlarmLog.Gone(Slot := _persistEvt);
    _persistEvt := 0;
END_IF
END_METHOD

// §3.8b — "restore is fail-closed and never silent". Every module that ran
// M_RestoreStationCfg and found an unrecognized image is holding one report;
// this takes them and annunciates each with the OWNING module's canonical path,
// which is what makes the message actionable instead of "something was lost".
//
// The event is AUTO_RESET and therefore never blocking: the consequence belongs
// to E_ConfigRestorePolicy, evaluated in ReleaseReportStart, so a station that
// declared DEFAULTS_AND_ANNUNCIATE really does run while the annunciation
// stands. It stays open until an ENGINEER acknowledges it, because nothing
// makes a lost image come back and an event that closed itself would be a lie.
METHOD PRIVATE _M_DrainRestoreLoss
VAR
    guard    : INT;
    path     : STRING(80);
    expected : UINT;
    found    : UINT;
END_VAR
// Bounded per scan (§5.6): losses are one-shot, so a large subtree simply
// finishes draining over the next few scans instead of stretching one.
FOR guard := 1 TO PL_Fraktal.MAX_EM_CHILDREN DO
    IF NOT M_TakeRestoreLoss(Path => path, Expected => expected, Found => found) THEN
        RETURN;
    END_IF
    ConfigPersist.RestoreLost := TRUE;
    ConfigPersist.RestoreAcknowledged := FALSE;
    ConfigPersist.LostPath := path;
    IF _restoreEvt = 0 THEN
        _restoreEvt := AlarmLog.Raise(Reason := E_Reason.CONFIG_RESTORE_LOST,
            Text := 'std.error.configRestoreLost', Source := path,
            Severity := E_Severity.MED, Category := E_Category.SYSTEM,
            ResetClass := E_ResetClass.AUTO_RESET);
    ELSE
        // A second losing module gets its own ring entry naming ITS path: a
        // summary that named only the first would hide the rest of the damage.
        _M_RaiseMaintenance(Reason := E_Reason.CONFIG_RESTORE_LOST,
            Text := 'std.error.configRestoreLost');
    END_IF
END_FOR
END_METHOD

// §3.8b — an operator of at least ENGINEER level accepts that a configuration
// image was lost. Under BLOCK_UNTIL_ACKNOWLEDGED this is what releases
// START_STOP again; under DEFAULTS_AND_ANNUNCIATE it is what clears the
// standing annunciation.
//
// The level is checked directly rather than through a gated action, because
// §3.8b names ENGINEER specifically and a station may legitimately have left
// DATA_WRITE or CONFIG_SET open to a lower level. Acknowledging a lost
// commissioning is a different decision from editing a value.
METHOD AcknowledgeConfigRestore : BOOL
AcknowledgeConfigRestore := FALSE;
IF Access.CurrentLevel < E_AccessLevel.ENGINEER THEN
    RETURN;
END_IF
IF NOT ConfigPersist.RestoreLost THEN
    RETURN;                                // nothing to acknowledge
END_IF
ConfigPersist.RestoreAcknowledged := TRUE;
IF _restoreEvt > 0 THEN
    AlarmLog.Gone(Slot := _restoreEvt);
    _restoreEvt := 0;
END_IF
Access.RecordActivity();
AcknowledgeConfigRestore := TRUE;
END_METHOD

// §3.8b — refuse a set operation, naming the offending record. "One rejection
// aborts the whole load naming the offending (Scope, WriteKey)": a refusal that
// says only "rejected" leaves an engineer diffing two machines by hand.
METHOD PRIVATE _M_RejectConfigSet
VAR_INPUT
    Scope : STRING(80);
    Key   : STRING(160);
END_VAR
ConfigPersist.LastRejectScope := Scope;
ConfigPersist.LastRejectKey := Key;
_M_RaiseMaintenance(Reason := E_Reason.CONFIG_SET_REJECTED,
    Text := 'std.error.configSetRejected');
END_METHOD

// §3.8b — the gate every set operation shares: CONFIG_SET (never DATA_WRITE —
// replacing a machine's entire parametrization is not the same decision as
// changing one number), a wired store, and the owning root READY.
METHOD PRIVATE _M_SetOpAllowed : BOOL
_M_SetOpAllowed := FALSE;
IF NOT Access.PermitsLogged(Gate := E_GatedAction.CONFIG_SET) THEN
    RETURN;
END_IF
IF _configStore = 0 THEN
    RETURN;
END_IF
IF _exec <> E_ExecState.READY THEN
    RETURN;
END_IF
_M_SetOpAllowed := TRUE;
END_METHOD

// §3.8b - remove a named set. Gated exactly like save and load (CONFIG_SET, a
// wired store, the root READY) because removing somebody's commissioned set is
// the same order of decision as replacing it, and audited with the set name.
// A store that has held MAX_CONFIG_SETS names needs this to hold a new one.
METHOD DeleteConfigSet : BOOL
VAR_INPUT
    SetName : STRING(80);
END_VAR
DeleteConfigSet := FALSE;
ConfigPersist.LastSetName := SetName;
ConfigPersist.LastSetRecords := 0;
IF NOT _M_SetOpAllowed() THEN
    RETURN;
END_IF
IF NOT _configStore.M_Delete(SetName := SetName) THEN
    RETURN;
END_IF
DeleteConfigSet := TRUE;
// The store's retained memory changed; not durable until written out.
_M_MarkPersistPending();
ListConfigSets();                          // the published listing follows
END_METHOD

// §3.8d - the effective level to read or write one registered value, from
// what its owning module declared and this root's policy. The root's own
// framework keys (unit.modePolicy.*) are in the built-in class. An unknown key
// resolves to ADMIN: the write path refuses it anyway, and a level check must
// never be the thing that lets an unknown key through.
METHOD PRIVATE _M_DataLevelOf : E_AccessLevel
VAR_INPUT
    TargetPath : STRING(255);
    WriteKey   : STRING(160);
    ForWrite   : BOOL;
END_VAR
VAR
    grant    : ST_ConfigAccess;
    minLevel : E_AccessLevel;
END_VAR
_M_DataLevelOf := E_AccessLevel.ADMIN;
IF (TargetPath = Status.Name) AND (LEFT(WriteKey, 16) = 'unit.modePolicy.') THEN
    _M_DataLevelOf := Access.M_DataLevel(ClassId := '', MinLevel := E_AccessLevel.NONE,
        ForWrite := ForWrite);
    RETURN;
END_IF
IF NOT M_ConfigAccessOf(Scope := TargetPath, WriteKey := WriteKey, Grant := grant) THEN
    RETURN;
END_IF
IF ForWrite THEN
    minLevel := grant.MinWriteLevel;
ELSE
    minLevel := grant.MinReadLevel;
END_IF
_M_DataLevelOf := Access.M_DataLevel(ClassId := grant.ClassId, MinLevel := minLevel,
    ForWrite := ForWrite);
END_METHOD

// §3.8d - declare a project data class on this root, at Setup. The levels are
// defaults: a class the deployment already edited keeps its persisted levels.
METHOD M_DeclareDataClass : BOOL
VAR_INPUT
    ClassId    : STRING(80);
    LabelKey   : STRING(160);
    ReadLevel  : E_AccessLevel;
    WriteLevel : E_AccessLevel;
END_VAR
M_DeclareDataClass := Access.M_DeclareClass(ClassId := ClassId,
    LabelKey := LabelKey, ReadLevel := ReadLevel, WriteLevel := WriteLevel);
END_METHOD

// §3.8d/§7.7(b) - edit a class's read or write level. The same gate as
// every other policy edit (ACCESS_POLICY), audited through the mailbox.
METHOD SetDataClassLevel : BOOL
VAR_INPUT
    ClassId  : STRING(160);
    Level    : DINT;
    ForWrite : BOOL;
END_VAR
VAR
    levelReq : E_AccessLevel;
END_VAR
SetDataClassLevel := FALSE;
IF NOT Access.PermitsLogged(Gate := E_GatedAction.ACCESS_POLICY) THEN
    RETURN;
END_IF
IF (Level < TO_DINT(E_AccessLevel.NONE)) OR (Level > TO_DINT(E_AccessLevel.ADMIN))
OR (LEN(ClassId) > 40) THEN
    RETURN;
END_IF
levelReq := Level;                          // range-checked above
SetDataClassLevel := Access.M_SetClassLevel(ClassId := ClassId,
    Level := levelReq, ForWrite := ForWrite);
IF SetDataClassLevel THEN
    ConfigRev := ConfigRev + 1;             // every manifest level may have moved
END_IF
END_METHOD

// §3.8e - TRUE when a (Scope, WriteKey) the subtree did not own names a value of
// the line this Unit references: the line is published under this Unit's own
// scope, and its keys alone begin 'line.'.
METHOD PRIVATE _M_IsLineKey : BOOL
VAR_INPUT
    Scope    : STRING(255);
    WriteKey : STRING(160);
END_VAR
_M_IsLineKey := (_pLine <> 0) AND (Scope = Status.Name)
    AND (LEFT(WriteKey, 5) = 'line.');
END_METHOD

// §3.8e - the subtree first; a line key it does not own goes to the line.
METHOD M_ApplyConfigWrite : BOOL
VAR_INPUT
    Scope     : STRING(255);
    WriteKey  : STRING(160);
    Revision  : UDINT;
    TextValue : STRING(255);
    RootReady : BOOL;
END_VAR
M_ApplyConfigWrite := SUPER^.M_ApplyConfigWrite(Scope := Scope,
    WriteKey := WriteKey, Revision := Revision, TextValue := TextValue,
    RootReady := RootReady);
IF (NOT M_ApplyConfigWrite) AND _M_IsLineKey(Scope := Scope, WriteKey := WriteKey) THEN
    M_ApplyConfigWrite := _pLine^.M_ApplyConfigWrite(Scope := _pLine^.Status.Name,
        WriteKey := WriteKey, Revision := Revision, TextValue := TextValue,
        RootReady := RootReady);
END_IF
END_METHOD

// §3.8e - the staging walk is the write walk, line leg included.
METHOD M_StageConfigWrite : BOOL
VAR_INPUT
    Scope     : STRING(255);
    WriteKey  : STRING(160);
    Revision  : UDINT;
    TextValue : STRING(255);
    RootReady : BOOL;
END_VAR
M_StageConfigWrite := SUPER^.M_StageConfigWrite(Scope := Scope,
    WriteKey := WriteKey, Revision := Revision, TextValue := TextValue,
    RootReady := RootReady);
IF (NOT M_StageConfigWrite) AND _M_IsLineKey(Scope := Scope, WriteKey := WriteKey) THEN
    M_StageConfigWrite := _pLine^.M_StageConfigWrite(Scope := _pLine^.Status.Name,
        WriteKey := WriteKey, Revision := Revision, TextValue := TextValue,
        RootReady := RootReady);
END_IF
END_METHOD

// §3.8e - the capture walk is the write walk, line leg included.
METHOD M_ApplyCapture : BOOL
VAR_INPUT
    Scope     : STRING(255);
    WriteKey  : STRING(160);
    Revision  : UDINT;
    RootReady : BOOL;
END_VAR
M_ApplyCapture := SUPER^.M_ApplyCapture(Scope := Scope, WriteKey := WriteKey,
    Revision := Revision, RootReady := RootReady);
IF (NOT M_ApplyCapture) AND _M_IsLineKey(Scope := Scope, WriteKey := WriteKey) THEN
    M_ApplyCapture := _pLine^.M_ApplyCapture(Scope := _pLine^.Status.Name,
        WriteKey := WriteKey, Revision := Revision, RootReady := RootReady);
END_IF
END_METHOD

// §3.8e/§3.8d - the access walk is the write walk, line leg included, so a line
// value is checked against the level the line declared for it.
METHOD M_ConfigAccessOf : BOOL
VAR_INPUT
    Scope    : STRING(255);
    WriteKey : STRING(160);
END_VAR
VAR_IN_OUT
    Grant : ST_ConfigAccess;
END_VAR
M_ConfigAccessOf := SUPER^.M_ConfigAccessOf(Scope := Scope, WriteKey := WriteKey,
    Grant := Grant);
IF (NOT M_ConfigAccessOf) AND _M_IsLineKey(Scope := Scope, WriteKey := WriteKey) THEN
    M_ConfigAccessOf := _pLine^.M_ConfigAccessOf(Scope := _pLine^.Status.Name,
        WriteKey := WriteKey, Grant := Grant);
END_IF
END_METHOD

// Core §3.8a - declare this root's own recipe record (its ParCfg) and the
// provider it is loaded from. The PAR_CFG values registered inside it become
// editable for EVERY model the root offers (AvailableModels), not only the
// active one, and an edit is written back to the provider's record so a
// changeover keeps it - when the provider is also an I_RecipeStore.
METHOD M_RegisterModelData : BOOL
VAR_INPUT
    pData     : PVOID;
    Size      : UDINT;
    RecipeKey : STRING(80);
    Provider  : I_RecipeProvider;
END_VAR
M_RegisterModelData := FALSE;
IF (pData = 0) OR (Size = 0) OR (Size > PL_Fraktal.MAX_MODEL_DATA_BYTES)
OR (RecipeKey = '') OR (Provider = 0) THEN
    RETURN;
END_IF
_modelProvider := Provider;
_modelKey := RecipeKey;
M_RegisterModelData := _M_SetModelRegion(pRegion := pData, Size := Size);
END_METHOD

// Serve model-scoped values of AvailableModels[Index] for this one request. 0,
// or the active model's index, is the live record and opens nothing. The record
// is loaded over a copy of the live one, so the provider's SchemaVersion check
// compares like with like. FALSE = no such model, or its record did not load.
METHOD PRIVATE _M_OpenModelView : BOOL
VAR_INPUT
    Index : UDINT;
END_VAR
_M_OpenModelView := FALSE;
_pModelView := 0;
_viewModelCode := '';
IF Index = 0 THEN
    _M_OpenModelView := TRUE;
    RETURN;
END_IF
IF (_modelProvider = 0) OR (_pModelRegion = 0)
OR (Index > TO_UDINT(AvailableModelCount)) THEN
    RETURN;
END_IF
IF AvailableModels[Index].ModelCode = Model.ModelCode THEN
    _M_OpenModelView := TRUE;              // the active model: its record is live
    RETURN;
END_IF
MEMCPY(destAddr := ADR(_modelBuf), srcAddr := _pModelRegion, n := _modelRegionSize);
IF NOT _modelProvider.Load(ModelCode := AvailableModels[Index].ModelCode,
        RecipeKey := _modelKey, pParCfg := ADR(_modelBuf), Size := _modelRegionSize) THEN
    RETURN;
END_IF
_viewModelCode := AvailableModels[Index].ModelCode;
_pModelView := ADR(_modelBuf);
_M_OpenModelView := TRUE;
END_METHOD

// §3.8a - WriteConfig for the model AvailableModels[ModelIndex] (0 = the active
// model). A model-data value is stored in that model's record and saved back to
// the provider; any other value is written as WriteConfig writes it.
METHOD WriteModelConfig : BOOL
VAR_INPUT
    ModelIndex : UDINT;
    TargetPath : STRING(255);
    WriteKey   : STRING(160);
    Revision   : DINT;
    TextValue  : STRING(255);
END_VAR
WriteModelConfig := FALSE;
IF NOT _M_OpenModelView(Index := ModelIndex) THEN
    RETURN;
END_IF
WriteModelConfig := WriteConfig(TargetPath := TargetPath, WriteKey := WriteKey,
    Revision := Revision, TextValue := TextValue);
_pModelView := 0;
END_METHOD

// §3.8a - the manifest walk (M_AppendConfig) with the model-data values of
// AvailableModels[ModelIndex] (0 = the active model). FALSE = no such model.
// For another model the walk yields that model's data only: the rest of the
// manifest is the running station's and is served by index 0.
METHOD M_AppendModelConfig : BOOL
VAR_INPUT
    Pager      : REFERENCE TO FB_ConfigPager;
    ModelIndex : UDINT;
END_VAR
M_AppendModelConfig := FALSE;
IF NOT _M_OpenModelView(Index := ModelIndex) THEN
    RETURN;
END_IF
Pager.M_SetModelOnly(Enabled := ModelIndex > 0);
M_AppendConfig(Pager := Pager);
Pager.M_SetModelOnly(Enabled := FALSE);
_pModelView := 0;
M_AppendModelConfig := TRUE;
END_METHOD

// Write the record a model-scoped value was just stored into back to the
// provider: the viewed model's buffer, or the live record for the active model.
METHOD PRIVATE _M_SaveModelData : BOOL
VAR
    store : I_RecipeStore;
END_VAR
_M_SaveModelData := FALSE;
IF _modelProvider = 0 THEN
    RETURN;
END_IF
IF NOT __QUERYINTERFACE(_modelProvider, store) THEN
    RETURN;
END_IF
IF _pModelView <> 0 THEN
    _M_SaveModelData := store.Save(ModelCode := _viewModelCode, RecipeKey := _modelKey,
        pData := _pModelView, Size := _modelRegionSize);
ELSE
    _M_SaveModelData := store.Save(ModelCode := Model.ModelCode, RecipeKey := _modelKey,
        pData := _pModelRegion, Size := _modelRegionSize);
END_IF
END_METHOD

// §3.8e/§8.5.2 - reference the line this root belongs to (owner or mirror, on
// this controller). A Unit references at most one line; 0 detaches it.
METHOD SetLine : BOOL
VAR_INPUT
    pLine : POINTER TO FB_LineData;
END_VAR
_pLine := pLine;
_lineHost := FALSE;
IF pLine <> 0 THEN
    // The first root to reference a line hosts it (ticks it, lends its log); a
    // line is never a child, so nothing else would run it (§3.8e(a)).
    _lineHost := pLine^.M_BindHost(pHost := THIS, pAlarmLog := ADR(AlarmLog));
END_IF
_shiftInit := FALSE;
CurrentShift := 0;
SetLine := (pLine <> 0);
END_METHOD

// §8.5.2(b) - evaluate the shift in force and close the one that just ended. Called
// every scan by the base with the synchronized clock; public so the SAME code can
// be driven across a boundary by a test instead of waiting for one. TRUE on the
// call that closed a shift.
METHOD M_ShiftTick : BOOL
VAR_INPUT
    Now          : DT;
    Synchronized : BOOL;
END_VAR
VAR
    idx : INT;
END_VAR
M_ShiftTick := FALSE;
IF _pLine = 0 THEN
    CurrentShift := 0;
    RETURN;
END_IF
idx := _pLine^.M_CurrentShift(MinuteOfDay := _pLine^.M_MinuteOfDay(Now := Now));
IF NOT _shiftInit THEN
    _shiftInit := TRUE;
    CurrentShift := idx;
    ShiftStartedAt := Now;
    _shiftSync := Synchronized;
    _shiftManualReset := FALSE;
    RETURN;
END_IF
IF idx = CurrentShift THEN
    RETURN;
END_IF
IF CurrentShift > 0 THEN
    _M_CloseShift(Now := Now, Synchronized := Synchronized);
    M_ShiftTick := TRUE;
END_IF
CurrentShift := idx;
ShiftStartedAt := Now;
_shiftSync := Synchronized;
_shiftManualReset := FALSE;
END_METHOD

// §8.5.2(b) - one operation in one scan: record the ending shift as its figures stood,
// then reset the per-shift counts and OEE accumulators (the trend ring is kept). A
// boundary on an unsynchronized clock still closes - stopping the accounting would
// lose more than a late boundary does - and the record says so.
METHOD PRIVATE _M_CloseShift
VAR_INPUT
    Now          : DT;
    Synchronized : BOOL;
END_VAR
VAR
    i         : INT;
    auditSlot : INT;
END_VAR
FOR i := PL_Fraktal.MAX_SHIFT_HISTORY TO 2 BY -1 DO
    ShiftHistory[i] := ShiftHistory[i - 1];
END_FOR
IF ShiftHistoryCount >= PL_Fraktal.MAX_SHIFT_HISTORY THEN
    ShiftHistoryTruncated := TRUE;
ELSE
    ShiftHistoryCount := ShiftHistoryCount + 1;
END_IF
ShiftHistory[1].ShiftIndex := CurrentShift;
ShiftHistory[1].StartAt := ShiftStartedAt;
ShiftHistory[1].EndAt := Now;
ShiftHistory[1].TimeSynchronized := _shiftSync AND Synchronized;
ShiftHistory[1].ManualReset := _shiftManualReset;
ShiftHistory[1].GoodCount := GoodCount;
ShiftHistory[1].NokCount := NokCount;
ShiftHistory[1].ReworkCount := ReworkCount;
ShiftHistory[1].RunMs := Oee.RunMs;
ShiftHistory[1].DownMs := Oee.DownMs;
ShiftHistory[1].IdleMs := Oee.IdleMs;
ShiftHistory[1].Availability := Oee.Availability;
ShiftHistory[1].AvailValid := Oee.AvailValid;
ShiftHistory[1].Performance := Oee.Performance;
ShiftHistory[1].PerfValid := Oee.PerfValid;
ShiftHistory[1].Quality := Oee.Quality;
ShiftHistory[1].QualValid := Oee.QualValid;
ShiftHistory[1].Oee := Oee.Oee;
ShiftHistory[1].OeeValid := Oee.OeeValid;
GoodCount := 0;
NokCount := 0;
ReworkCount := 0;
Oee.RunMs := 0;
Oee.DownMs := 0;
Oee.IdleMs := 0;
_M_OeeCompute();
auditSlot := AlarmLog.Raise(Reason := E_Reason.NONE, Text := 'std.audit.shiftClosed',
    Source := _name, Severity := E_Severity.LOW, Category := E_Category.SYSTEM,
    ResetClass := E_ResetClass.AUTO_RESET);
IF auditSlot > 0 THEN
    AlarmLog.Gone(Slot := auditSlot);    // come+gone: into the ring and the event sink
END_IF
END_METHOD

